LIN {X 0,Y 432.916,Z 623.479,A -85,B 0,C 180,E1 19556.175,E2 19556.175} C_VEL
LIN {X 0,Y 430.996,Z 639.731,A -85,B 0,C 180,E1 19554.827,E2 19554.827} C_VEL
LIN {X 0,Y 428.968,Z 654.603,A -85,B 0,C 180,E1 19553.313,E2 19553.313} C_VEL
LIN {X 0,Y 426.86,Z 668.614,A -85,B 0,C 180,E1 19551.576,E2 19551.576} C_VEL
LIN {X 0,Y 424.795,Z 681.338,A -85,B 0,C 180,E1 19549.668,E2 19549.668} C_VEL
LIN {X 0,Y 422.892,Z 692.644,A -85,B 0,C 180,E1 19547.615,E2 19547.615} C_VEL
LIN {X 0,Y 421.141,Z 703.114,A -85,B 0,C 180,E1 19545.279,E2 19545.279} C_VEL
LIN {X 0,Y 419.749,Z 711.572,A -85,B 0,C 180,E1 19542.939,E2 19542.939} C_VEL
LIN {X 0,Y 418.624,Z 718.946,A -85,B 0,C 180,E1 19540.319,E2 19540.319} C_VEL
LIN {X 0,Y 417.88,Z 724.436,A -85,B 0,C 180,E1 19537.7,E2 19537.7} C_VEL
LIN {X 0,Y 417.414,Z 728.221,A -85,B 0,C 180,E1 19535.085,E2 19535.085} C_VEL
LIN {X 0,Y 417.168,Z 730.486,A -85,B 0,C 180,E1 19532.335,E2 19532.335} C_VEL
LIN {X 0,Y 417.109,Z 731.085,A -85,B 0,C 180,E1 19529.588,E2 19529.588} C_VEL
LIN {X 0,Y 417.21,Z 730.043,A -85,B 0,C 180,E1 19526.84,E2 19526.84} C_VEL
LIN {X 0,Y 417.516,Z 727.312,A -85,B 0,C 180,E1 19524.09,E2 19524.09} C_VEL
LIN {X 0,Y 418.1,Z 722.784,A -85,B 0,C 180,E1 19521.335,E2 19521.335} C_VEL
LIN {X 0,Y 418.949,Z 716.685,A -85,B 0,C 180,E1 19518.715,E2 19518.715} C_VEL
LIN {X 0,Y 420.139,Z 709.085,A -85,B 0,C 180,E1 19516.233,E2 19516.233} C_VEL
LIN {X 0,Y 421.646,Z 700.029,A -85,B 0,C 180,E1 19513.893,E2 19513.893} C_VEL
LIN {X 0,Y 423.426,Z 689.42,A -85,B 0,C 180,E1 19511.672,E2 19511.672} C_VEL
LIN {X 0,Y 425.411,Z 677.603,A -85,B 0,C 180,E1 19509.645,E2 19509.645} C_VEL
LIN {X 0,Y 427.552,Z 664.114,A -85,B 0,C 180,E1 19507.738,E2 19507.738} C_VEL
LIN {X 0,Y 429.701,Z 649.518,A -85,B 0,C 180,E1 19506.045,E2 19506.045} C_VEL
LIN {X 0,Y 431.738,Z 633.856,A -85,B 0,C 180,E1 19504.559,E2 19504.559} C_VEL
LIN {X 0,Y 433.596,Z 617.11,A -85,B 0,C 180,E1 19503.279,E2 19503.279} C_VEL
LIN {X 0,Y 435.079,Z 600.265,A -85,B 0,C 180,E1 19502.26,E2 19502.26} C_VEL
LIN {X 0,Y 436.268,Z 581.748,A -85,B 0,C 180,E1 19501.409,E2 19501.409} C_VEL
LIN {X 0,Y 436.995,Z 563.024,A -85,B 0,C 180,E1 19500.806,E2 19500.806} C_VEL
LIN {X 0,Y 437.369,Z 538.708,A -85,B 0,C 180,E1 19500.338,E2 19500.338} C_VEL
LIN {X 0,Y 440.401,Z 366.683,A -85,B 0,C 180,E1 19497.558,E2 19497.558} C_VEL
LIN {X 0,Y 438.664,Z 359.169,A -85,B 0,C 180,E1 19497.254,E2 19497.254} C_VEL
LIN {X 0,Y 429.753,Z 342.969,A -85,B 0,C 180,E1 19496.041,E2 19496.041} C_VEL
LIN {X 0,Y 423.803,Z 326.84,A -85,B 0,C 180,E1 19493.336,E2 19493.336} C_VEL
LIN {X 0,Y 418.468,Z 313.652,A -85,B 0,C 180,E1 19490.893,E2 19490.893} C_VEL
LIN {X 0,Y 417.399,Z 310.595,A -85,B 0,C 180,E1 19490.241,E2 19490.241} C_VEL
LIN {X 0,Y 417.367,Z 310.446,A -85,B 0,C 180,E1 19486.343,E2 19486.343} C_VEL
LIN {X 0,Y 417.361,Z 310.494,A -85,B 0,C 180,E1 19482.452,E2 19482.452} C_VEL
LIN {X 0,Y 417.347,Z 310.491,A -85,B 0,C 180,E1 19478.649,E2 19478.649} C_VEL
LIN {X 0,Y 417.341,Z 310.491,A -85,B 0,C 180,E1 19474.764,E2 19474.764} C_VEL
LIN {X 0,Y 417.335,Z 310.495,A -85,B 0,C 180,E1 19470.845,E2 19470.845} C_VEL
LIN {X 0,Y 417.335,Z 310.499,A -85,B 0,C 180,E1 19466.924,E2 19466.924} C_VEL
LIN {X 0,Y 417.336,Z 310.498,A -85,B 0,C 180,E1 19463.079,E2 19463.079} C_VEL
LIN {X 0,Y 417.355,Z 310.477,A -85,B 0,C 180,E1 19459.451,E2 19459.451} C_VEL
LIN {X 0,Y 417.368,Z 310.483,A -85,B 0,C 180,E1 19455.564,E2 19455.564} C_VEL
LIN {X 0,Y 417.358,Z 310.496,A -85,B 0,C 180,E1 19451.75,E2 19451.75} C_VEL
LIN {X 0,Y 417.343,Z 310.478,A -85,B 0,C 180,E1 19447.849,E2 19447.849} C_VEL
LIN {X 0,Y 417.317,Z 310.49,A -85,B 0,C 180,E1 19444.122,E2 19444.122} C_VEL
LIN {X 0,Y 417.302,Z 310.501,A -85,B 0,C 180,E1 19440.412,E2 19440.412} C_VEL
LIN {X 0,Y 417.303,Z 310.484,A -85,B 0,C 180,E1 19436.566,E2 19436.566} C_VEL
LIN {X 0,Y 417.318,Z 310.487,A -85,B 0,C 180,E1 19432.843,E2 19432.843} C_VEL
LIN {X 0,Y 417.345,Z 310.499,A -85,B 0,C 180,E1 19429.09,E2 19429.09} C_VEL
LIN {X 0,Y 417.373,Z 310.483,A -85,B 0,C 180,E1 19425.29,E2 19425.29} C_VEL
LIN {X 0,Y 417.364,Z 310.479,A -85,B 0,C 180,E1 19421.421,E2 19421.421} C_VEL
LIN {X 0,Y 417.353,Z 310.485,A -85,B 0,C 180,E1 19417.61,E2 19417.61} C_VEL
LIN {X 0,Y 417.34,Z 310.493,A -85,B 0,C 180,E1 19413.844,E2 19413.844} C_VEL
LIN {X 0,Y 417.334,Z 310.497,A -85,B 0,C 180,E1 19410.111,E2 19410.111} C_VEL
LIN {X 0,Y 417.337,Z 310.486,A -85,B 0,C 180,E1 19406.233,E2 19406.233} C_VEL
LIN {X 0,Y 417.341,Z 310.465,A -85,B 0,C 180,E1 19402.344,E2 19402.344} C_VEL
LIN {X 0,Y 417.358,Z 310.451,A -85,B 0,C 180,E1 19398.608,E2 19398.608} C_VEL
LIN {X 0,Y 417.389,Z 310.785,A -85,B 0,C 180,E1 19398.001,E2 19398.001} C_VEL
LIN {X 0,Y 418.612,Z 313.856,A -85,B 0,C 180,E1 19397.472,E2 19397.472} C_VEL
LIN {X 0,Y 425.196,Z 327.627,A -85,B 0,C 180,E1 19395.324,E2 19395.324} C_VEL
LIN {X 0,Y 433.412,Z 346.345,A -85,B 0,C 180,E1 19392.705,E2 19392.705} C_VEL
LIN {X 0,Y 439.742,Z 362.777,A -85,B 0,C 180,E1 19390.648,E2 19390.648} C_VEL
LIN {X 0,Y 437.871,Z 383.994,A -85,B 0,C 180,E1 19389.058,E2 19389.058} C_VEL
LIN {X 0,Y 441.536,Z 419.357,A -85,B 0,C 180,E1 19387.995,E2 19387.995} C_VEL
LIN {X 0,Y 435.739,Z 636.384,A -85,B 0,C 180,E1 19384.015,E2 19384.015} C_VEL
LIN {X 0,Y 434.519,Z 657.893,A -85,B 0,C 180,E1 19383.442,E2 19383.442} C_VEL
LIN {X 0,Y 432.751,Z 679.3,A -85,B 0,C 180,E1 19382.622,E2 19382.622} C_VEL
LIN {X 0,Y 430.784,Z 699.969,A -85,B 0,C 180,E1 19381.559,E2 19381.559} C_VEL
LIN {X 0,Y 428.751,Z 719.018,A -85,B 0,C 180,E1 19380.323,E2 19380.323} C_VEL
LIN {X 0,Y 426.668,Z 737.44,A -85,B 0,C 180,E1 19378.864,E2 19378.864} C_VEL
LIN {X 0,Y 424.603,Z 755.114,A -85,B 0,C 180,E1 19377.182,E2 19377.182} C_VEL
LIN {X 0,Y 422.491,Z 773.079,A -85,B 0,C 180,E1 19375.137,E2 19375.137} C_VEL
LIN {X 0,Y 420.637,Z 789.749,A -85,B 0,C 180,E1 19372.869,E2 19372.869} C_VEL
LIN {X 0,Y 419.154,Z 804.214,A -85,B 0,C 180,E1 19370.527,E2 19370.527} C_VEL
LIN {X 0,Y 418.029,Z 816.771,A -85,B 0,C 180,E1 19368.115,E2 19368.115} C_VEL
LIN {X 0,Y 417.232,Z 827.882,A -85,B 0,C 180,E1 19365.568,E2 19365.568} C_VEL
LIN {X 0,Y 416.703,Z 837.456,A -85,B 0,C 180,E1 19362.894,E2 19362.894} C_VEL
LIN {X 0,Y 416.453,Z 845.052,A -85,B 0,C 180,E1 19360.234,E2 19360.234} C_VEL
LIN {X 0,Y 416.366,Z 850.572,A -85,B 0,C 180,E1 19357.728,E2 19357.728} C_VEL
LIN {X 0,Y 416.386,Z 854.593,A -85,B 0,C 180,E1 19355.097,E2 19355.097} C_VEL
LIN {X 0,Y 416.426,Z 856.966,A -85,B 0,C 180,E1 19352.477,E2 19352.477} C_VEL
LIN {X 0,Y 416.447,Z 857.743,A -85,B 0,C 180,E1 19349.862,E2 19349.862} C_VEL
LIN {X 0,Y 416.427,Z 856.813,A -85,B 0,C 180,E1 19347.248,E2 19347.248} C_VEL
LIN {X 0,Y 416.387,Z 854.237,A -85,B 0,C 180,E1 19344.627,E2 19344.627} C_VEL
LIN {X 0,Y 416.374,Z 850.01,A -85,B 0,C 180,E1 19341.994,E2 19341.994} C_VEL
LIN {X 0,Y 416.483,Z 844.036,A -85,B 0,C 180,E1 19339.348,E2 19339.348} C_VEL
LIN {X 0,Y 416.764,Z 836.113,A -85,B 0,C 180,E1 19336.685,E2 19336.685} C_VEL
LIN {X 0,Y 417.308,Z 826.752,A -85,B 0,C 180,E1 19334.149,E2 19334.149} C_VEL
LIN {X 0,Y 418.148,Z 815.386,A -85,B 0,C 180,E1 19331.602,E2 19331.602} C_VEL
LIN {X 0,Y 419.315,Z 802.509,A -85,B 0,C 180,E1 19329.183,E2 19329.183} C_VEL
LIN {X 0,Y 420.797,Z 788.255,A -85,B 0,C 180,E1 19326.918,E2 19326.918} C_VEL
LIN {X 0,Y 422.553,Z 772.476,A -85,B 0,C 180,E1 19324.792,E2 19324.792} C_VEL
LIN {X 0,Y 424.601,Z 755.097,A -85,B 0,C 180,E1 19322.818,E2 19322.818} C_VEL
LIN {X 0,Y 426.762,Z 736.64,A -85,B 0,C 180,E1 19321.067,E2 19321.067} C_VEL
LIN {X 0,Y 428.972,Z 717.108,A -85,B 0,C 180,E1 19319.54,E2 19319.54} C_VEL
LIN {X 0,Y 431.019,Z 697.589,A -85,B 0,C 180,E1 19318.304,E2 19318.304} C_VEL
LIN {X 0,Y 432.834,Z 678.286,A -85,B 0,C 180,E1 19317.335,E2 19317.335} C_VEL
LIN {X 0,Y 434.552,Z 657.279,A -85,B 0,C 180,E1 19316.541,E2 19316.541} C_VEL
LIN {X 0,Y 435.772,Z 635.074,A -85,B 0,C 180,E1 19315.961,E2 19315.961} C_VEL
LIN {X 0,Y 441.555,Z 417.909,A -85,B 0,C 180,E1 19311.983,E2 19311.983} C_VEL
LIN {X 0,Y 437.832,Z 382.808,A -85,B 0,C 180,E1 19310.888,E2 19310.888} C_VEL
LIN {X 0,Y 439.679,Z 362.43,A -85,B 0,C 180,E1 19309.323,E2 19309.323} C_VEL
LIN {X 0,Y 431.887,Z 342.744,A -85,B 0,C 180,E1 19306.824,E2 19306.824} C_VEL
LIN {X 0,Y 423.924,Z 324.867,A -85,B 0,C 180,E1 19304.278,E2 19304.278} C_VEL
LIN {X 0,Y 419.049,Z 314.463,A -85,B 0,C 180,E1 19302.658,E2 19302.658} C_VEL
LIN {X 0,Y 417.415,Z 310.928,A -85,B 0,C 180,E1 19302.052,E2 19302.052} C_VEL
LIN {X 0,Y 417.349,Z 310.452,A -85,B 0,C 180,E1 19301.576,E2 19301.576} C_VEL
LIN {X 0,Y 417.34,Z 310.47,A -85,B 0,C 180,E1 19297.83,E2 19297.83} C_VEL
LIN {X 0,Y 417.339,Z 310.481,A -85,B 0,C 180,E1 19293.932,E2 19293.932} C_VEL
LIN {X 0,Y 417.341,Z 310.495,A -85,B 0,C 180,E1 19290.047,E2 19290.047} C_VEL
LIN {X 0,Y 417.351,Z 310.49,A -85,B 0,C 180,E1 19286.309,E2 19286.309} C_VEL
LIN {X 0,Y 417.369,Z 310.482,A -85,B 0,C 180,E1 19282.538,E2 19282.538} C_VEL
LIN {X 0,Y 417.371,Z 310.479,A -85,B 0,C 180,E1 19278.724,E2 19278.724} C_VEL
LIN {X 0,Y 417.36,Z 310.488,A -85,B 0,C 180,E1 19274.853,E2 19274.853} C_VEL
LIN {X 0,Y 417.336,Z 310.499,A -85,B 0,C 180,E1 19271.05,E2 19271.05} C_VEL
LIN {X 0,Y 417.316,Z 310.489,A -85,B 0,C 180,E1 19267.295,E2 19267.295} C_VEL
LIN {X 0,Y 417.307,Z 310.487,A -85,B 0,C 180,E1 19263.571,E2 19263.571} C_VEL
LIN {X 0,Y 417.308,Z 310.502,A -85,B 0,C 180,E1 19259.725,E2 19259.725} C_VEL
LIN {X 0,Y 417.322,Z 310.486,A -85,B 0,C 180,E1 19256.016,E2 19256.016} C_VEL
LIN {X 0,Y 417.355,Z 310.478,A -85,B 0,C 180,E1 19252.29,E2 19252.29} C_VEL
LIN {X 0,Y 417.357,Z 310.5,A -85,B 0,C 180,E1 19248.39,E2 19248.39} C_VEL
LIN {X 0,Y 417.349,Z 310.483,A -85,B 0,C 180,E1 19244.578,E2 19244.578} C_VEL
LIN {X 0,Y 417.33,Z 310.482,A -85,B 0,C 180,E1 19240.838,E2 19240.838} C_VEL
LIN {X 0,Y 417.324,Z 310.5,A -85,B 0,C 180,E1 19237.161,E2 19237.161} C_VEL
LIN {X 0,Y 417.328,Z 310.499,A -85,B 0,C 180,E1 19233.229,E2 19233.229} C_VEL
LIN {X 0,Y 417.333,Z 310.494,A -85,B 0,C 180,E1 19229.325,E2 19229.325} C_VEL
LIN {X 0,Y 417.344,Z 310.488,A -85,B 0,C 180,E1 19225.499,E2 19225.499} C_VEL
LIN {X 0,Y 417.37,Z 310.484,A -85,B 0,C 180,E1 19221.789,E2 19221.789} C_VEL
LIN {X 0,Y 417.382,Z 310.485,A -85,B 0,C 180,E1 19217.953,E2 19217.953} C_VEL
LIN {X 0,Y 417.375,Z 310.446,A -85,B 0,C 180,E1 19214.054,E2 19214.054} C_VEL
LIN {X 0,Y 417.381,Z 310.473,A -85,B 0,C 180,E1 19210.12,E2 19210.12} C_VEL
LIN {X 0,Y 417.423,Z 310.821,A -85,B 0,C 180,E1 19209.56,E2 19209.56} C_VEL
LIN {X 0,Y 423.284,Z 325.515,A -85,B 0,C 180,E1 19206.796,E2 19206.796} C_VEL
LIN {X 0,Y 429.434,Z 342.168,A -85,B 0,C 180,E1 19203.971,E2 19203.971} C_VEL
LIN {X 0,Y 430.778,Z 344.992,A -85,B 0,C 180,E1 19203.685,E2 19203.685} C_VEL
LIN {X 0,Y 439.064,Z 360.282,A -85,B 0,C 180,E1 19202.586,E2 19202.586} C_VEL
LIN {X 0,Y 440.446,Z 368.261,A -85,B 0,C 180,E1 19202.307,E2 19202.307} C_VEL
LIN {X 0,Y 437.093,Z 558.617,A -85,B 0,C 180,E1 19199.21,E2 19199.21} C_VEL
LIN {X 0,Y 436.455,Z 577.921,A -85,B 0,C 180,E1 19198.644,E2 19198.644} C_VEL
LIN {X 0,Y 435.833,Z 589.062,A -85,B 0,C 180,E1 19198.193,E2 19198.193} C_VEL
LIN {X 0,Y 434.477,Z 596.631,A -85,B 0,C 180,E1 19197.912,E2 19197.912} C_VEL
LIN {X 0,Y 428.112,Z 614.037,A -85,B 0,C 180,E1 19197.327,E2 19197.327} C_VEL
LIN {X 0,Y 426.369,Z 620.792,A -85,B 0,C 180,E1 19196.95,E2 19196.95} C_VEL
LIN {X 0,Y 426.252,Z 621.745,A -85,B 0,C 180,E1 19196.885,E2 19196.885} C_VEL
LIN {X 0,Y 424.256,Z 638.214,A -85,B 0,C 180,E1 19195.548,E2 19195.548} C_VEL
LIN {X 0,Y 422.152,Z 653.265,A -85,B 0,C 180,E1 19194.04,E2 19194.04} C_VEL
LIN {X 0,Y 420.017,Z 666.865,A -85,B 0,C 180,E1 19192.388,E2 19192.388} C_VEL
LIN {X 0,Y 417.793,Z 680.072,A -85,B 0,C 180,E1 19190.45,E2 19190.45} C_VEL
LIN {X 0,Y 415.714,Z 691.783,A -85,B 0,C 180,E1 19188.365,E2 19188.365} C_VEL
LIN {X 0,Y 413.892,Z 702.067,A -85,B 0,C 180,E1 19186.129,E2 19186.129} C_VEL
LIN {X 0,Y 412.327,Z 710.951,A -85,B 0,C 180,E1 19183.747,E2 19183.747} C_VEL
LIN {X 0,Y 411.096,Z 718.401,A -85,B 0,C 180,E1 19181.22,E2 19181.22} C_VEL
LIN {X 0,Y 410.21,Z 724.366,A -85,B 0,C 180,E1 19178.55,E2 19178.55} C_VEL
LIN {X 0,Y 409.629,Z 728.578,A -85,B 0,C 180,E1 19175.884,E2 19175.884} C_VEL
LIN {X 0,Y 409.305,Z 731.277,A -85,B 0,C 180,E1 19173.081,E2 19173.081} C_VEL
LIN {X 0,Y 409.2,Z 732.293,A -85,B 0,C 180,E1 19170.28,E2 19170.28} C_VEL
LIN {X 0,Y 409.271,Z 731.67,A -85,B 0,C 180,E1 19167.48,E2 19167.48} C_VEL
LIN {X 0,Y 409.538,Z 729.386,A -85,B 0,C 180,E1 19164.677,E2 19164.677} C_VEL
LIN {X 0,Y 410.084,Z 725.347,A -85,B 0,C 180,E1 19161.871,E2 19161.871} C_VEL
LIN {X 0,Y 410.908,Z 719.743,A -85,B 0,C 180,E1 19159.201,E2 19159.201} C_VEL
LIN {X 0,Y 412.133,Z 712.22,A -85,B 0,C 180,E1 19156.532,E2 19156.532} C_VEL
LIN {X 0,Y 413.645,Z 703.643,A -85,B 0,C 180,E1 19154.149,E2 19154.149} C_VEL
LIN {X 0,Y 415.525,Z 692.986,A -85,B 0,C 180,E1 19151.772,E2 19151.772} C_VEL
LIN {X 0,Y 417.57,Z 681.528,A -85,B 0,C 180,E1 19149.685,E2 19149.685} C_VEL
LIN {X 0,Y 419.849,Z 668.093,A -85,B 0,C 180,E1 19147.677,E2 19147.677} C_VEL
LIN {X 0,Y 422.052,Z 654.11,A -85,B 0,C 180,E1 19145.954,E2 19145.954} C_VEL
LIN {X 0,Y 424.252,Z 638.461,A -85,B 0,C 180,E1 19144.377,E2 19144.377} C_VEL
LIN {X 0,Y 426.243,Z 622.169,A -85,B 0,C 180,E1 19143.049,E2 19143.049} C_VEL
LIN {X 0,Y 427.946,Z 604.675,A -85,B 0,C 180,E1 19141.916,E2 19141.916} C_VEL
LIN {X 0,Y 429.264,Z 586.618,A -85,B 0,C 180,E1 19141.022,E2 19141.022} C_VEL
LIN {X 0,Y 430.126,Z 567.98,A -85,B 0,C 180,E1 19140.359,E2 19140.359} C_VEL
LIN {X 0,Y 430.528,Z 548.32,A -85,B 0,C 180,E1 19139.919,E2 19139.919} C_VEL
LIN {X 0,Y 433.863,Z 368.04,A -85,B 0,C 180,E1 19136.96,E2 19136.96} C_VEL
LIN {X 0,Y 432.581,Z 362.846,A -85,B 0,C 180,E1 19136.736,E2 19136.736} C_VEL
LIN {X 0,Y 421.819,Z 343.427,A -85,B 0,C 180,E1 19135.218,E2 19135.218} C_VEL
LIN {X 0,Y 415.921,Z 327.808,A -85,B 0,C 180,E1 19132.496,E2 19132.496} C_VEL
LIN {X 0,Y 410.61,Z 314.728,A -85,B 0,C 180,E1 19129.996,E2 19129.996} C_VEL
LIN {X 0,Y 409.438,Z 311.625,A -85,B 0,C 180,E1 19129.307,E2 19129.307} C_VEL
LIN {X 0,Y 409.42,Z 311.437,A -85,B 0,C 180,E1 19125.488,E2 19125.488} C_VEL
LIN {X 0,Y 409.436,Z 311.472,A -85,B 0,C 180,E1 19121.624,E2 19121.624} C_VEL
LIN {X 0,Y 409.442,Z 311.47,A -85,B 0,C 180,E1 19117.803,E2 19117.803} C_VEL
LIN {X 0,Y 409.438,Z 311.468,A -85,B 0,C 180,E1 19113.834,E2 19113.834} C_VEL
LIN {X 0,Y 409.449,Z 311.466,A -85,B 0,C 180,E1 19109.879,E2 19109.879} C_VEL
LIN {X 0,Y 409.43,Z 311.474,A -85,B 0,C 180,E1 19105.921,E2 19105.921} C_VEL
LIN {X 0,Y 409.415,Z 311.487,A -85,B 0,C 180,E1 19102.092,E2 19102.092} C_VEL
LIN {X 0,Y 409.398,Z 311.479,A -85,B 0,C 180,E1 19098.217,E2 19098.217} C_VEL
LIN {X 0,Y 409.381,Z 311.466,A -85,B 0,C 180,E1 19094.426,E2 19094.426} C_VEL
LIN {X 0,Y 409.377,Z 311.487,A -85,B 0,C 180,E1 19090.555,E2 19090.555} C_VEL
LIN {X 0,Y 409.37,Z 311.489,A -85,B 0,C 180,E1 19086.592,E2 19086.592} C_VEL
LIN {X 0,Y 409.364,Z 311.468,A -85,B 0,C 180,E1 19082.64,E2 19082.64} C_VEL
LIN {X 0,Y 409.372,Z 311.482,A -85,B 0,C 180,E1 19078.881,E2 19078.881} C_VEL
LIN {X 0,Y 409.394,Z 311.487,A -85,B 0,C 180,E1 19075.097,E2 19075.097} C_VEL
LIN {X 0,Y 409.416,Z 311.465,A -85,B 0,C 180,E1 19071.291,E2 19071.291} C_VEL
LIN {X 0,Y 409.422,Z 311.467,A -85,B 0,C 180,E1 19067.304,E2 19067.304} C_VEL
LIN {X 0,Y 409.429,Z 311.483,A -85,B 0,C 180,E1 19063.398,E2 19063.398} C_VEL
LIN {X 0,Y 409.429,Z 311.486,A -85,B 0,C 180,E1 19059.411,E2 19059.411} C_VEL
LIN {X 0,Y 409.413,Z 311.481,A -85,B 0,C 180,E1 19055.624,E2 19055.624} C_VEL
LIN {X 0,Y 409.404,Z 311.479,A -85,B 0,C 180,E1 19051.838,E2 19051.838} C_VEL
LIN {X 0,Y 409.4,Z 311.482,A -85,B 0,C 180,E1 19047.997,E2 19047.997} C_VEL
LIN {X 0,Y 409.395,Z 311.433,A -85,B 0,C 180,E1 19044.116,E2 19044.116} C_VEL
LIN {X 0,Y 409.404,Z 311.469,A -85,B 0,C 180,E1 19040.219,E2 19040.219} C_VEL
LIN {X 0,Y 409.488,Z 311.753,A -85,B 0,C 180,E1 19038.979,E2 19038.979} C_VEL
LIN {X 0,Y 410.878,Z 315.161,A -85,B 0,C 180,E1 19038.369,E2 19038.369} C_VEL
LIN {X 0,Y 417.354,Z 328.537,A -85,B 0,C 180,E1 19036.183,E2 19036.183} C_VEL
LIN {X 0,Y 425.615,Z 347.272,A -85,B 0,C 180,E1 19033.456,E2 19033.456} C_VEL
LIN {X 0,Y 432.84,Z 365.718,A -85,B 0,C 180,E1 19031.063,E2 19031.063} C_VEL
LIN {X 0,Y 431.181,Z 383.563,A -85,B 0,C 180,E1 19029.707,E2 19029.707} C_VEL
LIN {X 0,Y 434.934,Z 420.487,A -85,B 0,C 180,E1 19028.574,E2 19028.574} C_VEL
LIN {X 0,Y 428.868,Z 635.975,A -85,B 0,C 180,E1 19024.566,E2 19024.566} C_VEL
LIN {X 0,Y 427.59,Z 657.284,A -85,B 0,C 180,E1 19023.986,E2 19023.986} C_VEL
LIN {X 0,Y 425.77,Z 678.267,A -85,B 0,C 180,E1 19023.172,E2 19023.172} C_VEL
LIN {X 0,Y 423.67,Z 699.069,A -85,B 0,C 180,E1 19022.088,E2 19022.088} C_VEL
LIN {X 0,Y 421.507,Z 718.264,A -85,B 0,C 180,E1 19020.821,E2 19020.821} C_VEL
LIN {X 0,Y 419.298,Z 736.613,A -85,B 0,C 180,E1 19019.342,E2 19019.342} C_VEL
LIN {X 0,Y 417.021,Z 754.9,A -85,B 0,C 180,E1 19017.563,E2 19017.563} C_VEL
LIN {X 0,Y 414.87,Z 772.149,A -85,B 0,C 180,E1 19015.556,E2 19015.556} C_VEL
LIN {X 0,Y 412.957,Z 788.311,A -85,B 0,C 180,E1 19013.315,E2 19013.315} C_VEL
LIN {X 0,Y 411.362,Z 802.783,A -85,B 0,C 180,E1 19010.934,E2 19010.934} C_VEL
LIN {X 0,Y 410.167,Z 815.378,A -85,B 0,C 180,E1 19008.475,E2 19008.475} C_VEL
LIN {X 0,Y 409.313,Z 826.523,A -85,B 0,C 180,E1 19005.878,E2 19005.878} C_VEL
LIN {X 0,Y 408.754,Z 836.131,A -85,B 0,C 180,E1 19003.149,E2 19003.149} C_VEL
LIN {X 0,Y 408.506,Z 843.761,A -85,B 0,C 180,E1 19000.435,E2 19000.435} C_VEL
LIN {X 0,Y 408.424,Z 849.304,A -85,B 0,C 180,E1 18997.879,E2 18997.879} C_VEL
LIN {X 0,Y 408.46,Z 853.36,A -85,B 0,C 180,E1 18995.196,E2 18995.196} C_VEL
LIN {X 0,Y 408.514,Z 855.759,A -85,B 0,C 180,E1 18992.525,E2 18992.525} C_VEL
LIN {X 0,Y 408.54,Z 856.558,A -85,B 0,C 180,E1 18990,E2 18990} C_VEL
LIN {X 0,Y 408.515,Z 855.681,A -85,B 0,C 180,E1 18987.335,E2 18987.335} C_VEL
LIN {X 0,Y 408.462,Z 853.181,A -85,B 0,C 180,E1 18984.663,E2 18984.663} C_VEL
LIN {X 0,Y 408.429,Z 849.023,A -85,B 0,C 180,E1 18981.979,E2 18981.979} C_VEL
LIN {X 0,Y 408.516,Z 843.427,A -85,B 0,C 180,E1 18979.423,E2 18979.423} C_VEL
LIN {X 0,Y 408.765,Z 835.93,A -85,B 0,C 180,E1 18976.786,E2 18976.786} C_VEL
LIN {X 0,Y 409.313,Z 826.523,A -85,B 0,C 180,E1 18974.122,E2 18974.122} C_VEL
LIN {X 0,Y 410.167,Z 815.376,A -85,B 0,C 180,E1 18971.525,E2 18971.525} C_VEL
LIN {X 0,Y 411.364,Z 802.779,A -85,B 0,C 180,E1 18969.066,E2 18969.066} C_VEL
LIN {X 0,Y 412.956,Z 788.304,A -85,B 0,C 180,E1 18966.685,E2 18966.685} C_VEL
LIN {X 0,Y 414.868,Z 772.131,A -85,B 0,C 180,E1 18964.444,E2 18964.444} C_VEL
LIN {X 0,Y 417.103,Z 754.217,A -85,B 0,C 180,E1 18962.365,E2 18962.365} C_VEL
LIN {X 0,Y 419.395,Z 735.81,A -85,B 0,C 180,E1 18960.587,E2 18960.587} C_VEL
LIN {X 0,Y 421.736,Z 716.344,A -85,B 0,C 180,E1 18959.039,E2 18959.039} C_VEL
LIN {X 0,Y 423.888,Z 696.913,A -85,B 0,C 180,E1 18957.787,E2 18957.787} C_VEL
LIN {X 0,Y 425.839,Z 677.437,A -85,B 0,C 180,E1 18956.794,E2 18956.794} C_VEL
LIN {X 0,Y 427.644,Z 656.33,A -85,B 0,C 180,E1 18955.986,E2 18955.986} C_VEL
LIN {X 0,Y 428.917,Z 634.217,A -85,B 0,C 180,E1 18955.401,E2 18955.401} C_VEL
LIN {X 0,Y 434.949,Z 419.079,A -85,B 0,C 180,E1 18951.405,E2 18951.405} C_VEL
LIN {X 0,Y 431.128,Z 382.442,A -85,B 0,C 180,E1 18950.245,E2 18950.245} C_VEL
LIN {X 0,Y 432.662,Z 365.234,A -85,B 0,C 180,E1 18948.883,E2 18948.883} C_VEL
LIN {X 0,Y 424.953,Z 345.751,A -85,B 0,C 180,E1 18946.344,E2 18946.344} C_VEL
LIN {X 0,Y 416.913,Z 327.6,A -85,B 0,C 180,E1 18943.685,E2 18943.685} C_VEL
LIN {X 0,Y 410.84,Z 315.109,A -85,B 0,C 180,E1 18941.636,E2 18941.636} C_VEL
LIN {X 0,Y 409.479,Z 311.692,A -85,B 0,C 180,E1 18941.019,E2 18941.019} C_VEL
LIN {X 0,Y 409.431,Z 311.437,A -85,B 0,C 180,E1 18937.098,E2 18937.098} C_VEL
LIN {X 0,Y 409.427,Z 311.484,A -85,B 0,C 180,E1 18933.163,E2 18933.163} C_VEL
LIN {X 0,Y 409.412,Z 311.489,A -85,B 0,C 180,E1 18929.328,E2 18929.328} C_VEL
LIN {X 0,Y 409.395,Z 311.49,A -85,B 0,C 180,E1 18925.612,E2 18925.612} C_VEL
LIN {X 0,Y 409.389,Z 311.485,A -85,B 0,C 180,E1 18921.791,E2 18921.791} C_VEL
LIN {X 0,Y 409.389,Z 311.474,A -85,B 0,C 180,E1 18917.922,E2 18917.922} C_VEL
LIN {X 0,Y 409.395,Z 311.468,A -85,B 0,C 180,E1 18914.136,E2 18914.136} C_VEL
LIN {X 0,Y 409.405,Z 311.484,A -85,B 0,C 180,E1 18910.269,E2 18910.269} C_VEL
LIN {X 0,Y 409.423,Z 311.48,A -85,B 0,C 180,E1 18906.45,E2 18906.45} C_VEL
LIN {X 0,Y 409.413,Z 311.464,A -85,B 0,C 180,E1 18902.519,E2 18902.519} C_VEL
LIN {X 0,Y 409.397,Z 311.481,A -85,B 0,C 180,E1 18898.74,E2 18898.74} C_VEL
LIN {X 0,Y 409.389,Z 311.486,A -85,B 0,C 180,E1 18894.815,E2 18894.815} C_VEL
LIN {X 0,Y 409.37,Z 311.466,A -85,B 0,C 180,E1 18891.148,E2 18891.148} C_VEL
LIN {X 0,Y 409.372,Z 311.487,A -85,B 0,C 180,E1 18887.301,E2 18887.301} C_VEL
LIN {X 0,Y 409.38,Z 311.488,A -85,B 0,C 180,E1 18883.396,E2 18883.396} C_VEL
LIN {X 0,Y 409.386,Z 311.473,A -85,B 0,C 180,E1 18879.558,E2 18879.558} C_VEL
LIN {X 0,Y 409.415,Z 311.468,A -85,B 0,C 180,E1 18875.93,E2 18875.93} C_VEL
LIN {X 0,Y 409.434,Z 311.48,A -85,B 0,C 180,E1 18872.038,E2 18872.038} C_VEL
LIN {X 0,Y 409.442,Z 311.486,A -85,B 0,C 180,E1 18868.165,E2 18868.165} C_VEL
LIN {X 0,Y 409.438,Z 311.488,A -85,B 0,C 180,E1 18864.167,E2 18864.167} C_VEL
LIN {X 0,Y 409.441,Z 311.487,A -85,B 0,C 180,E1 18860.222,E2 18860.222} C_VEL
LIN {X 0,Y 409.432,Z 311.48,A -85,B 0,C 180,E1 18856.282,E2 18856.282} C_VEL
LIN {X 0,Y 409.423,Z 311.449,A -85,B 0,C 180,E1 18852.377,E2 18852.377} C_VEL
LIN {X 0,Y 409.445,Z 311.68,A -85,B 0,C 180,E1 18850.554,E2 18850.554} C_VEL
LIN {X 0,Y 414.039,Z 322.964,A -85,B 0,C 180,E1 18848.294,E2 18848.294} C_VEL
LIN {X 0,Y 420.183,Z 338.961,A -85,B 0,C 180,E1 18845.412,E2 18845.412} C_VEL
LIN {X 0,Y 422.114,Z 344.155,A -85,B 0,C 180,E1 18844.601,E2 18844.601} C_VEL
LIN {X 0,Y 432.944,Z 363.641,A -85,B 0,C 180,E1 18843.111,E2 18843.111} C_VEL
LIN {X 0,Y 433.926,Z 369.853,A -85,B 0,C 180,E1 18842.897,E2 18842.897} C_VEL
LIN {X 0,Y 430.344,Z 559.389,A -85,B 0,C 180,E1 18839.769,E2 18839.769} C_VEL
LIN {X 0,Y 429.672,Z 578.718,A -85,B 0,C 180,E1 18839.195,E2 18839.195} C_VEL
LIN {X 0,Y 428.534,Z 597.005,A -85,B 0,C 180,E1 18838.403,E2 18838.403} C_VEL
LIN {X 0,Y 427.032,Z 614.436,A -85,B 0,C 180,E1 18837.392,E2 18837.392} C_VEL
LIN {X 0,Y 426.252,Z 621.745,A -85,B 0,C 180,E1 18836.885,E2 18836.885} C_VEL
LIN {X 0,Y 424.656,Z 628.618,A -85,B 0,C 180,E1 18836.446,E2 18836.446} C_VEL
LIN {X 0,Y 417.575,Z 644.654,A -85,B 0,C 180,E1 18835.446,E2 18835.446} C_VEL
LIN {X 0,Y 415.555,Z 650.949,A -85,B 0,C 180,E1 18834.887,E2 18834.887} C_VEL
LIN {X 0,Y 415.401,Z 651.806,A -85,B 0,C 180,E1 18834.795,E2 18834.795} C_VEL
LIN {X 0,Y 412.991,Z 666.63,A -85,B 0,C 180,E1 18833.016,E2 18833.016} C_VEL
LIN {X 0,Y 410.554,Z 680.506,A -85,B 0,C 180,E1 18830.977,E2 18830.977} C_VEL
LIN {X 0,Y 408.344,Z 692.341,A -85,B 0,C 180,E1 18828.857,E2 18828.857} C_VEL
LIN {X 0,Y 406.394,Z 702.736,A -85,B 0,C 180,E1 18826.582,E2 18826.582} C_VEL
LIN {X 0,Y 404.717,Z 711.718,A -85,B 0,C 180,E1 18824.157,E2 18824.157} C_VEL
LIN {X 0,Y 403.38,Z 719.26,A -85,B 0,C 180,E1 18821.582,E2 18821.582} C_VEL
LIN {X 0,Y 402.414,Z 725.309,A -85,B 0,C 180,E1 18818.861,E2 18818.861} C_VEL
LIN {X 0,Y 401.778,Z 729.602,A -85,B 0,C 180,E1 18816.143,E2 18816.143} C_VEL
LIN {X 0,Y 401.414,Z 732.379,A -85,B 0,C 180,E1 18813.284,E2 18813.284} C_VEL
LIN {X 0,Y 401.291,Z 733.474,A -85,B 0,C 180,E1 18810.428,E2 18810.428} C_VEL
LIN {X 0,Y 401.356,Z 732.933,A -85,B 0,C 180,E1 18807.573,E2 18807.573} C_VEL
LIN {X 0,Y 401.632,Z 730.734,A -85,B 0,C 180,E1 18804.715,E2 18804.715} C_VEL
LIN {X 0,Y 402.161,Z 727.017,A -85,B 0,C 180,E1 18801.997,E2 18801.997} C_VEL
LIN {X 0,Y 403.008,Z 721.566,A -85,B 0,C 180,E1 18799.258,E2 18799.258} C_VEL
LIN {X 0,Y 404.18,Z 714.745,A -85,B 0,C 180,E1 18796.7,E2 18796.7} C_VEL
LIN {X 0,Y 405.709,Z 706.499,A -85,B 0,C 180,E1 18794.271,E2 18794.271} C_VEL
LIN {X 0,Y 407.496,Z 696.925,A -85,B 0,C 180,E1 18791.992,E2 18791.992} C_VEL
LIN {X 0,Y 409.545,Z 686.041,A -85,B 0,C 180,E1 18789.866,E2 18789.866} C_VEL
LIN {X 0,Y 411.773,Z 673.823,A -85,B 0,C 180,E1 18787.892,E2 18787.892} C_VEL
LIN {X 0,Y 414.185,Z 659.608,A -85,B 0,C 180,E1 18785.999,E2 18785.999} C_VEL
LIN {X 0,Y 416.559,Z 644.23,A -85,B 0,C 180,E1 18784.327,E2 18784.327} C_VEL
LIN {X 0,Y 418.648,Z 628.546,A -85,B 0,C 180,E1 18782.938,E2 18782.938} C_VEL
LIN {X 0,Y 420.602,Z 610.906,A -85,B 0,C 180,E1 18781.69,E2 18781.69} C_VEL
LIN {X 0,Y 422.101,Z 593.095,A -85,B 0,C 180,E1 18780.716,E2 18780.716} C_VEL
LIN {X 0,Y 423.186,Z 574.271,A -85,B 0,C 180,E1 18779.962,E2 18779.962} C_VEL
LIN {X 0,Y 423.733,Z 555.053,A -85,B 0,C 180,E1 18779.452,E2 18779.452} C_VEL
LIN {X 0,Y 427.381,Z 369.434,A -85,B 0,C 180,E1 18776.345,E2 18776.345} C_VEL
LIN {X 0,Y 426.448,Z 366.302,A -85,B 0,C 180,E1 18776.189,E2 18776.189} C_VEL
LIN {X 0,Y 414.197,Z 344.558,A -85,B 0,C 180,E1 18774.441,E2 18774.441} C_VEL
LIN {X 0,Y 408.67,Z 330.049,A -85,B 0,C 180,E1 18771.868,E2 18771.868} C_VEL
LIN {X 0,Y 402.76,Z 315.929,A -85,B 0,C 180,E1 18769.053,E2 18769.053} C_VEL
LIN {X 0,Y 401.525,Z 312.649,A -85,B 0,C 180,E1 18768.329,E2 18768.329} C_VEL
LIN {X 0,Y 401.478,Z 312.44,A -85,B 0,C 180,E1 18764.582,E2 18764.582} C_VEL
LIN {X 0,Y 401.468,Z 312.467,A -85,B 0,C 180,E1 18760.732,E2 18760.732} C_VEL
LIN {X 0,Y 401.464,Z 312.469,A -85,B 0,C 180,E1 18756.886,E2 18756.886} C_VEL
LIN {X 0,Y 401.46,Z 312.468,A -85,B 0,C 180,E1 18752.884,E2 18752.884} C_VEL
LIN {X 0,Y 401.461,Z 312.46,A -85,B 0,C 180,E1 18749.055,E2 18749.055} C_VEL
LIN {X 0,Y 401.464,Z 312.456,A -85,B 0,C 180,E1 18745.207,E2 18745.207} C_VEL
LIN {X 0,Y 401.472,Z 312.47,A -85,B 0,C 180,E1 18741.322,E2 18741.322} C_VEL
LIN {X 0,Y 401.475,Z 312.475,A -85,B 0,C 180,E1 18737.389,E2 18737.389} C_VEL
LIN {X 0,Y 401.485,Z 312.452,A -85,B 0,C 180,E1 18733.539,E2 18733.539} C_VEL
LIN {X 0,Y 401.478,Z 312.454,A -85,B 0,C 180,E1 18729.534,E2 18729.534} C_VEL
LIN {X 0,Y 401.473,Z 312.478,A -85,B 0,C 180,E1 18725.718,E2 18725.718} C_VEL
LIN {X 0,Y 401.463,Z 312.459,A -85,B 0,C 180,E1 18721.713,E2 18721.713} C_VEL
LIN {X 0,Y 401.446,Z 312.457,A -85,B 0,C 180,E1 18717.859,E2 18717.859} C_VEL
LIN {X 0,Y 401.445,Z 312.478,A -85,B 0,C 180,E1 18713.996,E2 18713.996} C_VEL
LIN {X 0,Y 401.44,Z 312.473,A -85,B 0,C 180,E1 18710.105,E2 18710.105} C_VEL
LIN {X 0,Y 401.439,Z 312.456,A -85,B 0,C 180,E1 18706.249,E2 18706.249} C_VEL
LIN {X 0,Y 401.443,Z 312.465,A -85,B 0,C 180,E1 18702.311,E2 18702.311} C_VEL
LIN {X 0,Y 401.45,Z 312.476,A -85,B 0,C 180,E1 18698.37,E2 18698.37} C_VEL
LIN {X 0,Y 401.457,Z 312.477,A -85,B 0,C 180,E1 18694.478,E2 18694.478} C_VEL
LIN {X 0,Y 401.472,Z 312.476,A -85,B 0,C 180,E1 18690.619,E2 18690.619} C_VEL
LIN {X 0,Y 401.482,Z 312.473,A -85,B 0,C 180,E1 18686.778,E2 18686.778} C_VEL
LIN {X 0,Y 401.487,Z 312.424,A -85,B 0,C 180,E1 18682.835,E2 18682.835} C_VEL
LIN {X 0,Y 401.483,Z 312.6,A -85,B 0,C 180,E1 18680.087,E2 18680.087} C_VEL
LIN {X 0,Y 401.977,Z 314.409,A -85,B 0,C 180,E1 18679.706,E2 18679.706} C_VEL
LIN {X 0,Y 403.647,Z 317.225,A -85,B 0,C 180,E1 18679.161,E2 18679.161} C_VEL
LIN {X 0,Y 411.959,Z 334.831,A -85,B 0,C 180,E1 18676.234,E2 18676.234} C_VEL
LIN {X 0,Y 419.94,Z 353.216,A -85,B 0,C 180,E1 18673.531,E2 18673.531} C_VEL
LIN {X 0,Y 425.942,Z 368.781,A -85,B 0,C 180,E1 18671.484,E2 18671.484} C_VEL
LIN {X 0,Y 424.548,Z 383.134,A -85,B 0,C 180,E1 18670.377,E2 18670.377} C_VEL
LIN {X 0,Y 428.38,Z 421.538,A -85,B 0,C 180,E1 18669.173,E2 18669.173} C_VEL
LIN {X 0,Y 422.048,Z 635.401,A -85,B 0,C 180,E1 18665.138,E2 18665.138} C_VEL
LIN {X 0,Y 420.712,Z 656.561,A -85,B 0,C 180,E1 18664.553,E2 18664.553} C_VEL
LIN {X 0,Y 418.852,Z 677.103,A -85,B 0,C 180,E1 18663.746,E2 18663.746} C_VEL
LIN {X 0,Y 416.672,Z 697.503,A -85,B 0,C 180,E1 18662.677,E2 18662.677} C_VEL
LIN {X 0,Y 414.42,Z 716.6,A -85,B 0,C 180,E1 18661.407,E2 18661.407} C_VEL
LIN {X 0,Y 412.063,Z 735.036,A -85,B 0,C 180,E1 18659.909,E2 18659.909} C_VEL
LIN {X 0,Y 409.64,Z 753.382,A -85,B 0,C 180,E1 18658.103,E2 18658.103} C_VEL
LIN {X 0,Y 407.343,Z 770.726,A -85,B 0,C 180,E1 18656.055,E2 18656.055} C_VEL
LIN {X 0,Y 405.274,Z 787.072,A -85,B 0,C 180,E1 18653.752,E2 18653.752} C_VEL
LIN {X 0,Y 403.568,Z 801.573,A -85,B 0,C 180,E1 18651.322,E2 18651.322} C_VEL
LIN {X 0,Y 402.31,Z 814.007,A -85,B 0,C 180,E1 18648.849,E2 18648.849} C_VEL
LIN {X 0,Y 401.391,Z 825.185,A -85,B 0,C 180,E1 18646.199,E2 18646.199} C_VEL
LIN {X 0,Y 400.807,Z 834.827,A -85,B 0,C 180,E1 18643.414,E2 18643.414} C_VEL
LIN {X 0,Y 400.554,Z 842.489,A -85,B 0,C 180,E1 18640.644,E2 18640.644} C_VEL
LIN {X 0,Y 400.48,Z 848.054,A -85,B 0,C 180,E1 18638.037,E2 18638.037} C_VEL
LIN {X 0,Y 400.534,Z 852.136,A -85,B 0,C 180,E1 18635.299,E2 18635.299} C_VEL
LIN {X 0,Y 400.6,Z 854.552,A -85,B 0,C 180,E1 18632.575,E2 18632.575} C_VEL
LIN {X 0,Y 400.631,Z 855.357,A -85,B 0,C 180,E1 18630,E2 18630} C_VEL
LIN {X 0,Y 400.601,Z 854.551,A -85,B 0,C 180,E1 18627.425,E2 18627.425} C_VEL
LIN {X 0,Y 400.534,Z 852.135,A -85,B 0,C 180,E1 18624.701,E2 18624.701} C_VEL
LIN {X 0,Y 400.481,Z 848.055,A -85,B 0,C 180,E1 18621.963,E2 18621.963} C_VEL
LIN {X 0,Y 400.554,Z 842.493,A -85,B 0,C 180,E1 18619.356,E2 18619.356} C_VEL
LIN {X 0,Y 400.808,Z 834.829,A -85,B 0,C 180,E1 18616.586,E2 18616.586} C_VEL
LIN {X 0,Y 401.392,Z 825.183,A -85,B 0,C 180,E1 18613.801,E2 18613.801} C_VEL
LIN {X 0,Y 402.31,Z 814.003,A -85,B 0,C 180,E1 18611.151,E2 18611.151} C_VEL
LIN {X 0,Y 403.587,Z 801.368,A -85,B 0,C 180,E1 18608.643,E2 18608.643} C_VEL
LIN {X 0,Y 405.27,Z 787.067,A -85,B 0,C 180,E1 18606.249,E2 18606.249} C_VEL
LIN {X 0,Y 407.34,Z 770.711,A -85,B 0,C 180,E1 18603.946,E2 18603.946} C_VEL
LIN {X 0,Y 409.638,Z 753.353,A -85,B 0,C 180,E1 18601.896,E2 18601.896} C_VEL
LIN {X 0,Y 412.059,Z 734.996,A -85,B 0,C 180,E1 18600.091,E2 18600.091} C_VEL
LIN {X 0,Y 414.537,Z 715.605,A -85,B 0,C 180,E1 18598.521,E2 18598.521} C_VEL
LIN {X 0,Y 416.797,Z 696.261,A -85,B 0,C 180,E1 18597.252,E2 18597.252} C_VEL
LIN {X 0,Y 418.842,Z 677.041,A -85,B 0,C 180,E1 18596.255,E2 18596.255} C_VEL
LIN {X 0,Y 420.754,Z 655.774,A -85,B 0,C 180,E1 18595.425,E2 18595.425} C_VEL
LIN {X 0,Y 422.094,Z 633.713,A -85,B 0,C 180,E1 18594.83,E2 18594.83} C_VEL
LIN {X 0,Y 428.393,Z 420.054,A -85,B 0,C 180,E1 18590.805,E2 18590.805} C_VEL
LIN {X 0,Y 424.501,Z 381.848,A -85,B 0,C 180,E1 18589.564,E2 18589.564} C_VEL
LIN {X 0,Y 425.87,Z 368.617,A -85,B 0,C 180,E1 18588.499,E2 18588.499} C_VEL
LIN {X 0,Y 418.455,Z 349.723,A -85,B 0,C 180,E1 18585.989,E2 18585.989} C_VEL
LIN {X 0,Y 410.699,Z 332.17,A -85,B 0,C 180,E1 18583.356,E2 18583.356} C_VEL
LIN {X 0,Y 404.68,Z 319.763,A -85,B 0,C 180,E1 18581.276,E2 18581.276} C_VEL
LIN {X 0,Y 403.187,Z 316.439,A -85,B 0,C 180,E1 18580.708,E2 18580.708} C_VEL
LIN {X 0,Y 401.523,Z 312.834,A -85,B 0,C 180,E1 18580.034,E2 18580.034} C_VEL
LIN {X 0,Y 401.471,Z 312.461,A -85,B 0,C 180,E1 18579.61,E2 18579.61} C_VEL
LIN {X 0,Y 401.458,Z 312.421,A -85,B 0,C 180,E1 18575.718,E2 18575.718} C_VEL
LIN {X 0,Y 401.461,Z 312.469,A -85,B 0,C 180,E1 18571.869,E2 18571.869} C_VEL
LIN {X 0,Y 401.458,Z 312.467,A -85,B 0,C 180,E1 18567.919,E2 18567.919} C_VEL
LIN {X 0,Y 401.457,Z 312.468,A -85,B 0,C 180,E1 18563.951,E2 18563.951} C_VEL
LIN {X 0,Y 401.459,Z 312.474,A -85,B 0,C 180,E1 18560.102,E2 18560.102} C_VEL
LIN {X 0,Y 401.463,Z 312.479,A -85,B 0,C 180,E1 18556.197,E2 18556.197} C_VEL
LIN {X 0,Y 401.472,Z 312.461,A -85,B 0,C 180,E1 18552.367,E2 18552.367} C_VEL
LIN {X 0,Y 401.48,Z 312.452,A -85,B 0,C 180,E1 18548.449,E2 18548.449} C_VEL
LIN {X 0,Y 401.476,Z 312.469,A -85,B 0,C 180,E1 18544.571,E2 18544.571} C_VEL
LIN {X 0,Y 401.482,Z 312.471,A -85,B 0,C 180,E1 18540.57,E2 18540.57} C_VEL
LIN {X 0,Y 401.462,Z 312.453,A -85,B 0,C 180,E1 18536.536,E2 18536.536} C_VEL
LIN {X 0,Y 401.471,Z 312.459,A -85,B 0,C 180,E1 18532.559,E2 18532.559} C_VEL
LIN {X 0,Y 401.463,Z 312.478,A -85,B 0,C 180,E1 18528.653,E2 18528.653} C_VEL
LIN {X 0,Y 401.448,Z 312.459,A -85,B 0,C 180,E1 18524.84,E2 18524.84} C_VEL
LIN {X 0,Y 401.448,Z 312.46,A -85,B 0,C 180,E1 18520.957,E2 18520.957} C_VEL
LIN {X 0,Y 401.447,Z 312.478,A -85,B 0,C 180,E1 18517.136,E2 18517.136} C_VEL
LIN {X 0,Y 401.451,Z 312.477,A -85,B 0,C 180,E1 18513.205,E2 18513.205} C_VEL
LIN {X 0,Y 401.454,Z 312.472,A -85,B 0,C 180,E1 18509.23,E2 18509.23} C_VEL
LIN {X 0,Y 401.459,Z 312.467,A -85,B 0,C 180,E1 18505.272,E2 18505.272} C_VEL
LIN {X 0,Y 401.469,Z 312.466,A -85,B 0,C 180,E1 18501.444,E2 18501.444} C_VEL
LIN {X 0,Y 401.489,Z 312.466,A -85,B 0,C 180,E1 18497.699,E2 18497.699} C_VEL
LIN {X 0,Y 401.491,Z 312.42,A -85,B 0,C 180,E1 18493.763,E2 18493.763} C_VEL
LIN {X 0,Y 401.525,Z 312.728,A -85,B 0,C 180,E1 18491.528,E2 18491.528} C_VEL
LIN {X 0,Y 402.853,Z 316.073,A -85,B 0,C 180,E1 18490.8,E2 18490.8} C_VEL
LIN {X 0,Y 408.845,Z 330.583,A -85,B 0,C 180,E1 18487.924,E2 18487.924} C_VEL
LIN {X 0,Y 414.239,Z 344.647,A -85,B 0,C 180,E1 18485.449,E2 18485.449} C_VEL
LIN {X 0,Y 426.584,Z 366.634,A -85,B 0,C 180,E1 18483.687,E2 18483.687} C_VEL
LIN {X 0,Y 427.461,Z 371.054,A -85,B 0,C 180,E1 18483.512,E2 18483.512} C_VEL
LIN {X 0,Y 423.636,Z 560.134,A -85,B 0,C 180,E1 18480.345,E2 18480.345} C_VEL
LIN {X 0,Y 422.93,Z 579.467,A -85,B 0,C 180,E1 18479.765,E2 18479.765} C_VEL
LIN {X 0,Y 421.763,Z 597.411,A -85,B 0,C 180,E1 18478.981,E2 18478.981} C_VEL
LIN {X 0,Y 420.184,Z 615,A -85,B 0,C 180,E1 18477.954,E2 18477.954} C_VEL
LIN {X 0,Y 418.23,Z 631.776,A -85,B 0,C 180,E1 18476.708,E2 18476.708} C_VEL
LIN {X 0,Y 416.059,Z 647.549,A -85,B 0,C 180,E1 18475.249,E2 18475.249} C_VEL
LIN {X 0,Y 415.401,Z 651.806,A -85,B 0,C 180,E1 18474.795,E2 18474.795} C_VEL
LIN {X 0,Y 413.589,Z 657.941,A -85,B 0,C 180,E1 18474.181,E2 18474.181} C_VEL
LIN {X 0,Y 406.154,Z 672.262,A -85,B 0,C 180,E1 18472.777,E2 18472.777} C_VEL
LIN {X 0,Y 404.023,Z 677.673,A -85,B 0,C 180,E1 18472.053,E2 18472.053} C_VEL
LIN {X 0,Y 403.855,Z 678.401,A -85,B 0,C 180,E1 18471.937,E2 18471.937} C_VEL
LIN {X 0,Y 401.456,Z 690.73,A -85,B 0,C 180,E1 18469.798,E2 18469.798} C_VEL
LIN {X 0,Y 399.286,Z 701.631,A -85,B 0,C 180,E1 18467.487,E2 18467.487} C_VEL
LIN {X 0,Y 397.364,Z 711.344,A -85,B 0,C 180,E1 18464.931,E2 18464.931} C_VEL
LIN {X 0,Y 395.898,Z 719.007,A -85,B 0,C 180,E1 18462.396,E2 18462.396} C_VEL
LIN {X 0,Y 394.773,Z 725.428,A -85,B 0,C 180,E1 18459.623,E2 18459.623} C_VEL
LIN {X 0,Y 394.021,Z 730.07,A -85,B 0,C 180,E1 18456.85,E2 18456.85} C_VEL
LIN {X 0,Y 393.572,Z 733.178,A -85,B 0,C 180,E1 18453.933,E2 18453.933} C_VEL
LIN {X 0,Y 393.392,Z 734.595,A -85,B 0,C 180,E1 18451.019,E2 18451.019} C_VEL
LIN {X 0,Y 393.423,Z 734.376,A -85,B 0,C 180,E1 18448.107,E2 18448.107} C_VEL
LIN {X 0,Y 393.666,Z 732.51,A -85,B 0,C 180,E1 18445.192,E2 18445.192} C_VEL
LIN {X 0,Y 394.166,Z 729.146,A -85,B 0,C 180,E1 18442.421,E2 18442.421} C_VEL
LIN {X 0,Y 394.99,Z 724.109,A -85,B 0,C 180,E1 18439.647,E2 18439.647} C_VEL
LIN {X 0,Y 396.186,Z 717.445,A -85,B 0,C 180,E1 18436.946,E2 18436.946} C_VEL
LIN {X 0,Y 397.767,Z 709.334,A -85,B 0,C 180,E1 18434.398,E2 18434.398} C_VEL
LIN {X 0,Y 399.711,Z 699.492,A -85,B 0,C 180,E1 18431.931,E2 18431.931} C_VEL
LIN {X 0,Y 401.973,Z 688.118,A -85,B 0,C 180,E1 18429.621,E2 18429.621} C_VEL
LIN {X 0,Y 404.292,Z 676.096,A -85,B 0,C 180,E1 18427.614,E2 18427.614} C_VEL
LIN {X 0,Y 406.707,Z 662.704,A -85,B 0,C 180,E1 18425.761,E2 18425.761} C_VEL
LIN {X 0,Y 409.156,Z 647.802,A -85,B 0,C 180,E1 18424.065,E2 18424.065} C_VEL
LIN {X 0,Y 411.335,Z 632.67,A -85,B 0,C 180,E1 18422.652,E2 18422.652} C_VEL
LIN {X 0,Y 413.382,Z 615.861,A -85,B 0,C 180,E1 18421.387,E2 18421.387} C_VEL
LIN {X 0,Y 415.07,Z 597.887,A -85,B 0,C 180,E1 18420.329,E2 18420.329} C_VEL
LIN {X 0,Y 416.304,Z 579.433,A -85,B 0,C 180,E1 18419.522,E2 18419.522} C_VEL
LIN {X 0,Y 417.013,Z 560.547,A -85,B 0,C 180,E1 18418.955,E2 18418.955} C_VEL
LIN {X 0,Y 420.97,Z 370.964,A -85,B 0,C 180,E1 18415.716,E2 18415.716} C_VEL
LIN {X 0,Y 408.892,Z 349.416,A -85,B 0,C 180,E1 18413.948,E2 18413.948} C_VEL
LIN {X 0,Y 406.12,Z 344.736,A -85,B 0,C 180,E1 18413.498,E2 18413.498} C_VEL
LIN {X 0,Y 400.354,Z 329.96,A -85,B 0,C 180,E1 18410.734,E2 18410.734} C_VEL
LIN {X 0,Y 394.968,Z 317.07,A -85,B 0,C 180,E1 18408.064,E2 18408.064} C_VEL
LIN {X 0,Y 393.56,Z 313.603,A -85,B 0,C 180,E1 18407.242,E2 18407.242} C_VEL
LIN {X 0,Y 393.548,Z 313.459,A -85,B 0,C 180,E1 18403.513,E2 18403.513} C_VEL
LIN {X 0,Y 393.558,Z 313.465,A -85,B 0,C 180,E1 18399.62,E2 18399.62} C_VEL
LIN {X 0,Y 393.554,Z 313.463,A -85,B 0,C 180,E1 18395.614,E2 18395.614} C_VEL
LIN {X 0,Y 393.552,Z 313.464,A -85,B 0,C 180,E1 18391.559,E2 18391.559} C_VEL
LIN {X 0,Y 393.559,Z 313.459,A -85,B 0,C 180,E1 18387.706,E2 18387.706} C_VEL
LIN {X 0,Y 393.556,Z 313.446,A -85,B 0,C 180,E1 18383.667,E2 18383.667} C_VEL
LIN {X 0,Y 393.55,Z 313.44,A -85,B 0,C 180,E1 18379.749,E2 18379.749} C_VEL
LIN {X 0,Y 393.547,Z 313.451,A -85,B 0,C 180,E1 18375.775,E2 18375.775} C_VEL
LIN {X 0,Y 393.531,Z 313.462,A -85,B 0,C 180,E1 18371.877,E2 18371.877} C_VEL
LIN {X 0,Y 393.522,Z 313.442,A -85,B 0,C 180,E1 18367.886,E2 18367.886} C_VEL
LIN {X 0,Y 393.503,Z 313.452,A -85,B 0,C 180,E1 18364.08,E2 18364.08} C_VEL
LIN {X 0,Y 393.488,Z 313.468,A -85,B 0,C 180,E1 18360.291,E2 18360.291} C_VEL
LIN {X 0,Y 393.488,Z 313.45,A -85,B 0,C 180,E1 18356.358,E2 18356.358} C_VEL
LIN {X 0,Y 393.492,Z 313.448,A -85,B 0,C 180,E1 18352.408,E2 18352.408} C_VEL
LIN {X 0,Y 393.501,Z 313.467,A -85,B 0,C 180,E1 18348.42,E2 18348.42} C_VEL
LIN {X 0,Y 393.504,Z 313.467,A -85,B 0,C 180,E1 18344.36,E2 18344.36} C_VEL
LIN {X 0,Y 393.509,Z 313.457,A -85,B 0,C 180,E1 18340.404,E2 18340.404} C_VEL
LIN {X 0,Y 393.516,Z 313.45,A -85,B 0,C 180,E1 18336.49,E2 18336.49} C_VEL
LIN {X 0,Y 393.525,Z 313.449,A -85,B 0,C 180,E1 18332.621,E2 18332.621} C_VEL
LIN {X 0,Y 393.542,Z 313.449,A -85,B 0,C 180,E1 18328.782,E2 18328.782} C_VEL
LIN {X 0,Y 393.549,Z 313.409,A -85,B 0,C 180,E1 18324.891,E2 18324.891} C_VEL
LIN {X 0,Y 393.602,Z 313.683,A -85,B 0,C 180,E1 18321.138,E2 18321.138} C_VEL
LIN {X 0,Y 394.75,Z 316.793,A -85,B 0,C 180,E1 18320.524,E2 18320.524} C_VEL
LIN {X 0,Y 395.956,Z 318.911,A -85,B 0,C 180,E1 18320.104,E2 18320.104} C_VEL
LIN {X 0,Y 401.799,Z 330.761,A -85,B 0,C 180,E1 18317.98,E2 18317.98} C_VEL
LIN {X 0,Y 409.797,Z 348.447,A -85,B 0,C 180,E1 18315.161,E2 18315.161} C_VEL
LIN {X 0,Y 417.495,Z 367.578,A -85,B 0,C 180,E1 18312.471,E2 18312.471} C_VEL
LIN {X 0,Y 419.039,Z 372.186,A -85,B 0,C 180,E1 18311.888,E2 18311.888} C_VEL
LIN {X 0,Y 417.954,Z 382.538,A -85,B 0,C 180,E1 18311.074,E2 18311.074} C_VEL
LIN {X 0,Y 421.871,Z 422.728,A -85,B 0,C 180,E1 18309.787,E2 18309.787} C_VEL
LIN {X 0,Y 415.256,Z 635.275,A -85,B 0,C 180,E1 18305.721,E2 18305.721} C_VEL
LIN {X 0,Y 413.844,Z 656.322,A -85,B 0,C 180,E1 18305.123,E2 18305.123} C_VEL
LIN {X 0,Y 411.921,Z 676.513,A -85,B 0,C 180,E1 18304.314,E2 18304.314} C_VEL
LIN {X 0,Y 409.615,Z 696.882,A -85,B 0,C 180,E1 18303.229,E2 18303.229} C_VEL
LIN {X 0,Y 407.252,Z 715.888,A -85,B 0,C 180,E1 18301.942,E2 18301.942} C_VEL
LIN {X 0,Y 404.765,Z 734.249,A -85,B 0,C 180,E1 18300.423,E2 18300.423} C_VEL
LIN {X 0,Y 402.21,Z 752.538,A -85,B 0,C 180,E1 18298.589,E2 18298.589} C_VEL
LIN {X 0,Y 399.787,Z 769.779,A -85,B 0,C 180,E1 18296.514,E2 18296.514} C_VEL
LIN {X 0,Y 397.601,Z 785.904,A -85,B 0,C 180,E1 18294.198,E2 18294.198} C_VEL
LIN {X 0,Y 395.835,Z 799.983,A -85,B 0,C 180,E1 18291.796,E2 18291.796} C_VEL
LIN {X 0,Y 394.463,Z 812.649,A -85,B 0,C 180,E1 18289.239,E2 18289.239} C_VEL
LIN {X 0,Y 393.476,Z 823.859,A -85,B 0,C 180,E1 18286.535,E2 18286.535} C_VEL
LIN {X 0,Y 392.863,Z 833.534,A -85,B 0,C 180,E1 18283.691,E2 18283.691} C_VEL
LIN {X 0,Y 392.593,Z 841.224,A -85,B 0,C 180,E1 18280.863,E2 18280.863} C_VEL
LIN {X 0,Y 392.532,Z 847.083,A -85,B 0,C 180,E1 18278.053,E2 18278.053} C_VEL
LIN {X 0,Y 392.606,Z 851.096,A -85,B 0,C 180,E1 18275.26,E2 18275.26} C_VEL
LIN {X 0,Y 392.687,Z 853.424,A -85,B 0,C 180,E1 18272.481,E2 18272.481} C_VEL
LIN {X 0,Y 392.717,Z 854.138,A -85,B 0,C 180,E1 18269.854,E2 18269.854} C_VEL
LIN {X 0,Y 392.683,Z 853.267,A -85,B 0,C 180,E1 18267.227,E2 18267.227} C_VEL
LIN {X 0,Y 392.601,Z 850.733,A -85,B 0,C 180,E1 18264.447,E2 18264.447} C_VEL
LIN {X 0,Y 392.534,Z 846.526,A -85,B 0,C 180,E1 18261.652,E2 18261.652} C_VEL
LIN {X 0,Y 392.597,Z 840.885,A -85,B 0,C 180,E1 18258.989,E2 18258.989} C_VEL
LIN {X 0,Y 392.864,Z 833.534,A -85,B 0,C 180,E1 18256.309,E2 18256.309} C_VEL
LIN {X 0,Y 393.477,Z 823.854,A -85,B 0,C 180,E1 18253.465,E2 18253.465} C_VEL
LIN {X 0,Y 394.464,Z 812.641,A -85,B 0,C 180,E1 18250.761,E2 18250.761} C_VEL
LIN {X 0,Y 395.833,Z 799.971,A -85,B 0,C 180,E1 18248.204,E2 18248.204} C_VEL
LIN {X 0,Y 397.6,Z 785.884,A -85,B 0,C 180,E1 18245.802,E2 18245.802} C_VEL
LIN {X 0,Y 399.785,Z 769.75,A -85,B 0,C 180,E1 18243.486,E2 18243.486} C_VEL
LIN {X 0,Y 402.303,Z 751.833,A -85,B 0,C 180,E1 18241.337,E2 18241.337} C_VEL
LIN {X 0,Y 404.863,Z 733.507,A -85,B 0,C 180,E1 18239.511,E2 18239.511} C_VEL
LIN {X 0,Y 407.504,Z 713.952,A -85,B 0,C 180,E1 18237.914,E2 18237.914} C_VEL
LIN {X 0,Y 409.943,Z 694.091,A -85,B 0,C 180,E1 18236.607,E2 18236.607} C_VEL
LIN {X 0,Y 412.077,Z 674.905,A -85,B 0,C 180,E1 18235.617,E2 18235.617} C_VEL
LIN {X 0,Y 414.012,Z 653.942,A -85,B 0,C 180,E1 18234.802,E2 18234.802} C_VEL
LIN {X 0,Y 415.363,Z 632.112,A -85,B 0,C 180,E1 18234.215,E2 18234.215} C_VEL
LIN {X 0,Y 421.873,Z 421.052,A -85,B 0,C 180,E1 18230.186,E2 18230.186} C_VEL
LIN {X 0,Y 417.909,Z 381.477,A -85,B 0,C 180,E1 18228.879,E2 18228.879} C_VEL
LIN {X 0,Y 419.038,Z 371.813,A -85,B 0,C 180,E1 18228.081,E2 18228.081} C_VEL
LIN {X 0,Y 411.753,Z 353.239,A -85,B 0,C 180,E1 18225.554,E2 18225.554} C_VEL
LIN {X 0,Y 404.51,Z 336.713,A -85,B 0,C 180,E1 18223.016,E2 18223.016} C_VEL
LIN {X 0,Y 397.474,Z 321.825,A -85,B 0,C 180,E1 18220.466,E2 18220.466} C_VEL
LIN {X 0,Y 393.692,Z 314.172,A -85,B 0,C 180,E1 18219.033,E2 18219.033} C_VEL
LIN {X 0,Y 393.562,Z 313.469,A -85,B 0,C 180,E1 18218.68,E2 18218.68} C_VEL
LIN {X 0,Y 393.552,Z 313.417,A -85,B 0,C 180,E1 18214.687,E2 18214.687} C_VEL
LIN {X 0,Y 393.565,Z 313.448,A -85,B 0,C 180,E1 18210.706,E2 18210.706} C_VEL
LIN {X 0,Y 393.558,Z 313.448,A -85,B 0,C 180,E1 18206.723,E2 18206.723} C_VEL
LIN {X 0,Y 393.565,Z 313.444,A -85,B 0,C 180,E1 18202.715,E2 18202.715} C_VEL
LIN {X 0,Y 393.55,Z 313.443,A -85,B 0,C 180,E1 18198.67,E2 18198.67} C_VEL
LIN {X 0,Y 393.554,Z 313.448,A -85,B 0,C 180,E1 18194.717,E2 18194.717} C_VEL
LIN {X 0,Y 393.541,Z 313.466,A -85,B 0,C 180,E1 18190.688,E2 18190.688} C_VEL
LIN {X 0,Y 393.548,Z 313.454,A -85,B 0,C 180,E1 18186.608,E2 18186.608} C_VEL
LIN {X 0,Y 393.531,Z 313.44,A -85,B 0,C 180,E1 18182.621,E2 18182.621} C_VEL
LIN {X 0,Y 393.522,Z 313.456,A -85,B 0,C 180,E1 18178.689,E2 18178.689} C_VEL
LIN {X 0,Y 393.515,Z 313.464,A -85,B 0,C 180,E1 18174.751,E2 18174.751} C_VEL
LIN {X 0,Y 393.501,Z 313.442,A -85,B 0,C 180,E1 18170.936,E2 18170.936} C_VEL
LIN {X 0,Y 393.499,Z 313.457,A -85,B 0,C 180,E1 18167.079,E2 18167.079} C_VEL
LIN {X 0,Y 393.502,Z 313.467,A -85,B 0,C 180,E1 18163.162,E2 18163.162} C_VEL
LIN {X 0,Y 393.505,Z 313.455,A -85,B 0,C 180,E1 18159.162,E2 18159.162} C_VEL
LIN {X 0,Y 393.507,Z 313.444,A -85,B 0,C 180,E1 18155.213,E2 18155.213} C_VEL
LIN {X 0,Y 393.513,Z 313.453,A -85,B 0,C 180,E1 18151.231,E2 18151.231} C_VEL
LIN {X 0,Y 393.518,Z 313.46,A -85,B 0,C 180,E1 18147.235,E2 18147.235} C_VEL
LIN {X 0,Y 393.524,Z 313.464,A -85,B 0,C 180,E1 18143.338,E2 18143.338} C_VEL
LIN {X 0,Y 393.535,Z 313.458,A -85,B 0,C 180,E1 18139.426,E2 18139.426} C_VEL
LIN {X 0,Y 393.538,Z 313.431,A -85,B 0,C 180,E1 18135.474,E2 18135.474} C_VEL
LIN {X 0,Y 393.567,Z 313.66,A -85,B 0,C 180,E1 18132.613,E2 18132.613} C_VEL
LIN {X 0,Y 398.812,Z 326.272,A -85,B 0,C 180,E1 18129.899,E2 18129.899} C_VEL
LIN {X 0,Y 404.332,Z 340.049,A -85,B 0,C 180,E1 18127.225,E2 18127.225} C_VEL
LIN {X 0,Y 406.421,Z 345.401,A -85,B 0,C 180,E1 18126.322,E2 18126.322} C_VEL
LIN {X 0,Y 417.747,Z 365.108,A -85,B 0,C 180,E1 18124.638,E2 18124.638} C_VEL
LIN {X 0,Y 421.06,Z 371.655,A -85,B 0,C 180,E1 18124.156,E2 18124.156} C_VEL
LIN {X 0,Y 416.97,Z 560.855,A -85,B 0,C 180,E1 18120.941,E2 18120.941} C_VEL
LIN {X 0,Y 416.238,Z 580.043,A -85,B 0,C 180,E1 18120.36,E2 18120.36} C_VEL
LIN {X 0,Y 414.951,Z 598.933,A -85,B 0,C 180,E1 18119.521,E2 18119.521} C_VEL
LIN {X 0,Y 413.27,Z 616.635,A -85,B 0,C 180,E1 18118.464,E2 18118.464} C_VEL
LIN {X 0,Y 411.226,Z 633.289,A -85,B 0,C 180,E1 18117.2,E2 18117.2} C_VEL
LIN {X 0,Y 408.847,Z 649.658,A -85,B 0,C 180,E1 18115.649,E2 18115.649} C_VEL
LIN {X 0,Y 406.337,Z 664.754,A -85,B 0,C 180,E1 18113.884,E2 18113.884} C_VEL
LIN {X 0,Y 403.855,Z 678.401,A -85,B 0,C 180,E1 18111.937,E2 18111.937} C_VEL
LIN {X 0,Y 401.943,Z 683.676,A -85,B 0,C 180,E1 18111.153,E2 18111.153} C_VEL
LIN {X 0,Y 393.99,Z 696.367,A -85,B 0,C 180,E1 18109.222,E2 18109.222} C_VEL
LIN {X 0,Y 392.177,Z 700.714,A -85,B 0,C 180,E1 18108.337,E2 18108.337} C_VEL
LIN {X 0,Y 390.193,Z 710.225,A -85,B 0,C 180,E1 18105.913,E2 18105.913} C_VEL
LIN {X 0,Y 388.465,Z 718.608,A -85,B 0,C 180,E1 18103.242,E2 18103.242} C_VEL
LIN {X 0,Y 387.22,Z 725.118,A -85,B 0,C 180,E1 18100.564,E2 18100.564} C_VEL
LIN {X 0,Y 386.334,Z 730.204,A -85,B 0,C 180,E1 18097.734,E2 18097.734} C_VEL
LIN {X 0,Y 385.788,Z 733.618,A -85,B 0,C 180,E1 18094.906,E2 18094.906} C_VEL
LIN {X 0,Y 385.519,Z 735.537,A -85,B 0,C 180,E1 18091.932,E2 18091.932} C_VEL
LIN {X 0,Y 385.481,Z 735.811,A -85,B 0,C 180,E1 18088.96,E2 18088.96} C_VEL
LIN {X 0,Y 385.669,Z 734.451,A -85,B 0,C 180,E1 18085.986,E2 18085.986} C_VEL
LIN {X 0,Y 386.108,Z 731.587,A -85,B 0,C 180,E1 18083.159,E2 18083.159} C_VEL
LIN {X 0,Y 386.879,Z 727.097,A -85,B 0,C 180,E1 18080.329,E2 18080.329} C_VEL
LIN {X 0,Y 388.037,Z 720.843,A -85,B 0,C 180,E1 18077.5,E2 18077.5} C_VEL
LIN {X 0,Y 389.611,Z 713.082,A -85,B 0,C 180,E1 18074.826,E2 18074.826} C_VEL
LIN {X 0,Y 391.536,Z 703.858,A -85,B 0,C 180,E1 18072.309,E2 18072.309} C_VEL
LIN {X 0,Y 393.775,Z 693.191,A -85,B 0,C 180,E1 18069.954,E2 18069.954} C_VEL
LIN {X 0,Y 396.276,Z 681.051,A -85,B 0,C 180,E1 18067.762,E2 18067.762} C_VEL
LIN {X 0,Y 398.813,Z 667.874,A -85,B 0,C 180,E1 18065.802,E2 18065.802} C_VEL
LIN {X 0,Y 401.423,Z 653.145,A -85,B 0,C 180,E1 18064,E2 18064} C_VEL
LIN {X 0,Y 403.781,Z 638.127,A -85,B 0,C 180,E1 18062.496,E2 18062.496} C_VEL
LIN {X 0,Y 406.017,Z 621.425,A -85,B 0,C 180,E1 18061.141,E2 18061.141} C_VEL
LIN {X 0,Y 407.797,Z 604.816,A -85,B 0,C 180,E1 18060.07,E2 18060.07} C_VEL
LIN {X 0,Y 409.272,Z 586.2,A -85,B 0,C 180,E1 18059.155,E2 18059.155} C_VEL
LIN {X 0,Y 410.213,Z 566.946,A -85,B 0,C 180,E1 18058.489,E2 18058.489} C_VEL
LIN {X 0,Y 410.706,Z 542.868,A -85,B 0,C 180,E1 18057.988,E2 18057.988} C_VEL
LIN {X 0,Y 414.637,Z 373.964,A -85,B 0,C 180,E1 18055.1,E2 18055.1} C_VEL
LIN {X 0,Y 403.294,Z 353.738,A -85,B 0,C 180,E1 18053.385,E2 18053.385} C_VEL
LIN {X 0,Y 398.148,Z 345.046,A -85,B 0,C 180,E1 18052.52,E2 18052.52} C_VEL
LIN {X 0,Y 391.902,Z 329.245,A -85,B 0,C 180,E1 18049.416,E2 18049.416} C_VEL
LIN {X 0,Y 387.041,Z 318.11,A -85,B 0,C 180,E1 18046.978,E2 18046.978} C_VEL
LIN {X 0,Y 385.647,Z 314.605,A -85,B 0,C 180,E1 18046.118,E2 18046.118} C_VEL
LIN {X 0,Y 385.622,Z 314.44,A -85,B 0,C 180,E1 18042.138,E2 18042.138} C_VEL
LIN {X 0,Y 385.621,Z 314.435,A -85,B 0,C 180,E1 18038.105,E2 18038.105} C_VEL
LIN {X 0,Y 385.615,Z 314.434,A -85,B 0,C 180,E1 18034.061,E2 18034.061} C_VEL
LIN {X 0,Y 385.617,Z 314.433,A -85,B 0,C 180,E1 18030.003,E2 18030.003} C_VEL
LIN {X 0,Y 385.599,Z 314.444,A -85,B 0,C 180,E1 18026.156,E2 18026.156} C_VEL
LIN {X 0,Y 385.588,Z 314.455,A -85,B 0,C 180,E1 18022.226,E2 18022.226} C_VEL
LIN {X 0,Y 385.578,Z 314.444,A -85,B 0,C 180,E1 18018.287,E2 18018.287} C_VEL
LIN {X 0,Y 385.566,Z 314.43,A -85,B 0,C 180,E1 18014.416,E2 18014.416} C_VEL
LIN {X 0,Y 385.563,Z 314.453,A -85,B 0,C 180,E1 18010.459,E2 18010.459} C_VEL
LIN {X 0,Y 385.555,Z 314.456,A -85,B 0,C 180,E1 18006.552,E2 18006.552} C_VEL
LIN {X 0,Y 385.548,Z 314.432,A -85,B 0,C 180,E1 18002.527,E2 18002.527} C_VEL
LIN {X 0,Y 385.547,Z 314.444,A -85,B 0,C 180,E1 17998.514,E2 17998.514} C_VEL
LIN {X 0,Y 385.554,Z 314.456,A -85,B 0,C 180,E1 17994.494,E2 17994.494} C_VEL
LIN {X 0,Y 385.558,Z 314.445,A -85,B 0,C 180,E1 17990.447,E2 17990.447} C_VEL
LIN {X 0,Y 385.561,Z 314.432,A -85,B 0,C 180,E1 17986.351,E2 17986.351} C_VEL
LIN {X 0,Y 385.566,Z 314.441,A -85,B 0,C 180,E1 17982.338,E2 17982.338} C_VEL
LIN {X 0,Y 385.572,Z 314.449,A -85,B 0,C 180,E1 17978.234,E2 17978.234} C_VEL
LIN {X 0,Y 385.579,Z 314.451,A -85,B 0,C 180,E1 17974.131,E2 17974.131} C_VEL
LIN {X 0,Y 385.58,Z 314.45,A -85,B 0,C 180,E1 17970.14,E2 17970.14} C_VEL
LIN {X 0,Y 385.581,Z 314.427,A -85,B 0,C 180,E1 17966.076,E2 17966.076} C_VEL
LIN {X 0,Y 385.606,Z 314.558,A -85,B 0,C 180,E1 17962.365,E2 17962.365} C_VEL
LIN {X 0,Y 386.069,Z 316.334,A -85,B 0,C 180,E1 17961.948,E2 17961.948} C_VEL
LIN {X 0,Y 387.999,Z 319.736,A -85,B 0,C 180,E1 17961.23,E2 17961.23} C_VEL
LIN {X 0,Y 394.474,Z 332.948,A -85,B 0,C 180,E1 17958.776,E2 17958.776} C_VEL
LIN {X 0,Y 402.152,Z 349.684,A -85,B 0,C 180,E1 17955.98,E2 17955.98} C_VEL
LIN {X 0,Y 409.948,Z 368.876,A -85,B 0,C 180,E1 17953.176,E2 17953.176} C_VEL
LIN {X 0,Y 412.124,Z 375.317,A -85,B 0,C 180,E1 17952.316,E2 17952.316} C_VEL
LIN {X 0,Y 411.447,Z 382.221,A -85,B 0,C 180,E1 17951.784,E2 17951.784} C_VEL
LIN {X 0,Y 415.419,Z 423.705,A -85,B 0,C 180,E1 17950.425,E2 17950.425} C_VEL
LIN {X 0,Y 408.519,Z 634.944,A -85,B 0,C 180,E1 17946.328,E2 17946.328} C_VEL
LIN {X 0,Y 407.039,Z 655.856,A -85,B 0,C 180,E1 17945.721,E2 17945.721} C_VEL
LIN {X 0,Y 405.023,Z 676.041,A -85,B 0,C 180,E1 17944.896,E2 17944.896} C_VEL
LIN {X 0,Y 402.603,Z 696.28,A -85,B 0,C 180,E1 17943.799,E2 17943.799} C_VEL
LIN {X 0,Y 399.99,Z 716.125,A -85,B 0,C 180,E1 17942.423,E2 17942.423} C_VEL
LIN {X 0,Y 397.388,Z 734.247,A -85,B 0,C 180,E1 17940.881,E2 17940.881} C_VEL
LIN {X 0,Y 394.81,Z 751.702,A -85,B 0,C 180,E1 17939.093,E2 17939.093} C_VEL
LIN {X 0,Y 392.246,Z 768.898,A -85,B 0,C 180,E1 17936.982,E2 17936.982} C_VEL
LIN {X 0,Y 389.928,Z 784.982,A -85,B 0,C 180,E1 17934.625,E2 17934.625} C_VEL
LIN {X 0,Y 388.003,Z 799.438,A -85,B 0,C 180,E1 17932.1,E2 17932.1} C_VEL
LIN {X 0,Y 386.562,Z 811.997,A -85,B 0,C 180,E1 17929.491,E2 17929.491} C_VEL
LIN {X 0,Y 385.527,Z 823.11,A -85,B 0,C 180,E1 17926.73,E2 17926.73} C_VEL
LIN {X 0,Y 384.897,Z 832.698,A -85,B 0,C 180,E1 17923.827,E2 17923.827} C_VEL
LIN {X 0,Y 384.626,Z 840.306,A -85,B 0,C 180,E1 17920.939,E2 17920.939} C_VEL
LIN {X 0,Y 384.583,Z 845.847,A -85,B 0,C 180,E1 17918.221,E2 17918.221} C_VEL
LIN {X 0,Y 384.675,Z 849.795,A -85,B 0,C 180,E1 17915.437,E2 17915.437} C_VEL
LIN {X 0,Y 384.771,Z 852.141,A -85,B 0,C 180,E1 17912.681,E2 17912.681} C_VEL
LIN {X 0,Y 384.812,Z 852.954,A -85,B 0,C 180,E1 17910,E2 17910} C_VEL
LIN {X 0,Y 384.772,Z 852.14,A -85,B 0,C 180,E1 17907.319,E2 17907.319} C_VEL
LIN {X 0,Y 384.673,Z 849.694,A -85,B 0,C 180,E1 17904.481,E2 17904.481} C_VEL
LIN {X 0,Y 384.583,Z 845.846,A -85,B 0,C 180,E1 17901.779,E2 17901.779} C_VEL
LIN {X 0,Y 384.632,Z 839.966,A -85,B 0,C 180,E1 17898.909,E2 17898.909} C_VEL
LIN {X 0,Y 384.897,Z 832.697,A -85,B 0,C 180,E1 17896.173,E2 17896.173} C_VEL
LIN {X 0,Y 385.527,Z 823.103,A -85,B 0,C 180,E1 17893.27,E2 17893.27} C_VEL
LIN {X 0,Y 386.562,Z 811.985,A -85,B 0,C 180,E1 17890.509,E2 17890.509} C_VEL
LIN {X 0,Y 388.003,Z 799.422,A -85,B 0,C 180,E1 17887.9,E2 17887.9} C_VEL
LIN {X 0,Y 389.927,Z 784.958,A -85,B 0,C 180,E1 17885.375,E2 17885.375} C_VEL
LIN {X 0,Y 392.244,Z 768.864,A -85,B 0,C 180,E1 17883.017,E2 17883.017} C_VEL
LIN {X 0,Y 394.897,Z 751.073,A -85,B 0,C 180,E1 17880.839,E2 17880.839} C_VEL
LIN {X 0,Y 397.624,Z 732.652,A -85,B 0,C 180,E1 17878.971,E2 17878.971} C_VEL
LIN {X 0,Y 400.293,Z 713.881,A -85,B 0,C 180,E1 17877.407,E2 17877.407} C_VEL
LIN {X 0,Y 402.784,Z 694.725,A -85,B 0,C 180,E1 17876.111,E2 17876.111} C_VEL
LIN {X 0,Y 405.099,Z 675.163,A -85,B 0,C 180,E1 17875.068,E2 17875.068} C_VEL
LIN {X 0,Y 407.181,Z 653.862,A -85,B 0,C 180,E1 17874.217,E2 17874.217} C_VEL
LIN {X 0,Y 408.624,Z 631.863,A -85,B 0,C 180,E1 17873.61,E2 17873.61} C_VEL
LIN {X 0,Y 415.42,Z 422.205,A -85,B 0,C 180,E1 17869.553,E2 17869.553} C_VEL
LIN {X 0,Y 411.396,Z 380.893,A -85,B 0,C 180,E1 17868.154,E2 17868.154} C_VEL
LIN {X 0,Y 412.119,Z 374.753,A -85,B 0,C 180,E1 17867.625,E2 17867.625} C_VEL
LIN {X 0,Y 404.692,Z 355.738,A -85,B 0,C 180,E1 17864.959,E2 17864.959} C_VEL
LIN {X 0,Y 397.175,Z 338.608,A -85,B 0,C 180,E1 17862.233,E2 17862.233} C_VEL
LIN {X 0,Y 389.71,Z 323.102,A -85,B 0,C 180,E1 17859.445,E2 17859.445} C_VEL
LIN {X 0,Y 387.178,Z 318.289,A -85,B 0,C 180,E1 17858.489,E2 17858.489} C_VEL
LIN {X 0,Y 385.625,Z 314.681,A -85,B 0,C 180,E1 17857.727,E2 17857.727} C_VEL
LIN {X 0,Y 385.601,Z 314.41,A -85,B 0,C 180,E1 17854.458,E2 17854.458} C_VEL
LIN {X 0,Y 385.614,Z 314.439,A -85,B 0,C 180,E1 17850.544,E2 17850.544} C_VEL
LIN {X 0,Y 385.611,Z 314.438,A -85,B 0,C 180,E1 17846.552,E2 17846.552} C_VEL
LIN {X 0,Y 385.614,Z 314.434,A -85,B 0,C 180,E1 17842.566,E2 17842.566} C_VEL
LIN {X 0,Y 385.609,Z 314.431,A -85,B 0,C 180,E1 17838.598,E2 17838.598} C_VEL
LIN {X 0,Y 385.615,Z 314.434,A -85,B 0,C 180,E1 17834.567,E2 17834.567} C_VEL
LIN {X 0,Y 385.6,Z 314.451,A -85,B 0,C 180,E1 17830.457,E2 17830.457} C_VEL
LIN {X 0,Y 385.6,Z 314.446,A -85,B 0,C 180,E1 17826.401,E2 17826.401} C_VEL
LIN {X 0,Y 385.589,Z 314.429,A -85,B 0,C 180,E1 17822.378,E2 17822.378} C_VEL
LIN {X 0,Y 385.593,Z 314.44,A -85,B 0,C 180,E1 17818.514,E2 17818.514} C_VEL
LIN {X 0,Y 385.594,Z 314.456,A -85,B 0,C 180,E1 17814.345,E2 17814.345} C_VEL
LIN {X 0,Y 385.592,Z 314.431,A -85,B 0,C 180,E1 17810.447,E2 17810.447} C_VEL
LIN {X 0,Y 385.607,Z 314.428,A -85,B 0,C 180,E1 17806.352,E2 17806.352} C_VEL
LIN {X 0,Y 385.607,Z 314.448,A -85,B 0,C 180,E1 17802.339,E2 17802.339} C_VEL
LIN {X 0,Y 385.621,Z 314.448,A -85,B 0,C 180,E1 17798.236,E2 17798.236} C_VEL
LIN {X 0,Y 385.611,Z 314.436,A -85,B 0,C 180,E1 17794.121,E2 17794.121} C_VEL
LIN {X 0,Y 385.629,Z 314.431,A -85,B 0,C 180,E1 17790.144,E2 17790.144} C_VEL
LIN {X 0,Y 385.618,Z 314.434,A -85,B 0,C 180,E1 17786.067,E2 17786.067} C_VEL
LIN {X 0,Y 385.625,Z 314.435,A -85,B 0,C 180,E1 17782.017,E2 17782.017} C_VEL
LIN {X 0,Y 385.624,Z 314.438,A -85,B 0,C 180,E1 17778.013,E2 17778.013} C_VEL
LIN {X 0,Y 385.626,Z 314.47,A -85,B 0,C 180,E1 17773.879,E2 17773.879} C_VEL
LIN {X 0,Y 385.859,Z 315.653,A -85,B 0,C 180,E1 17773.485,E2 17773.485} C_VEL
LIN {X 0,Y 389.443,Z 323.771,A -85,B 0,C 180,E1 17771.658,E2 17771.658} C_VEL
LIN {X 0,Y 394.691,Z 336.105,A -85,B 0,C 180,E1 17769.075,E2 17769.075} C_VEL
LIN {X 0,Y 398.547,Z 345.9,A -85,B 0,C 180,E1 17767.259,E2 17767.259} C_VEL
LIN {X 0,Y 410.134,Z 365.728,A -85,B 0,C 180,E1 17765.461,E2 17765.461} C_VEL
LIN {X 0,Y 414.661,Z 374.464,A -85,B 0,C 180,E1 17764.781,E2 17764.781} C_VEL
LIN {X 0,Y 410.35,Z 561.559,A -85,B 0,C 180,E1 17761.555,E2 17761.555} C_VEL
LIN {X 0,Y 409.587,Z 580.645,A -85,B 0,C 180,E1 17760.971,E2 17760.971} C_VEL
LIN {X 0,Y 408.262,Z 599.362,A -85,B 0,C 180,E1 17760.135,E2 17760.135} C_VEL
LIN {X 0,Y 406.502,Z 617.193,A -85,B 0,C 180,E1 17759.063,E2 17759.063} C_VEL
LIN {X 0,Y 404.361,Z 633.932,A -85,B 0,C 180,E1 17757.781,E2 17757.781} C_VEL
LIN {X 0,Y 401.982,Z 649.691,A -85,B 0,C 180,E1 17756.278,E2 17756.278} C_VEL
LIN {X 0,Y 399.332,Z 665.051,A -85,B 0,C 180,E1 17754.48,E2 17754.48} C_VEL
LIN {X 0,Y 396.734,Z 678.706,A -85,B 0,C 180,E1 17752.524,E2 17752.524} C_VEL
LIN {X 0,Y 394.177,Z 691.263,A -85,B 0,C 180,E1 17750.335,E2 17750.335} C_VEL
LIN {X 0,Y 392.177,Z 700.714,A -85,B 0,C 180,E1 17748.337,E2 17748.337} C_VEL
LIN {X 0,Y 390.401,Z 704.945,A -85,B 0,C 180,E1 17747.419,E2 17747.419} C_VEL
LIN {X 0,Y 383.096,Z 714.504,A -85,B 0,C 180,E1 17745.235,E2 17745.235} C_VEL
LIN {X 0,Y 381.201,Z 717.867,A -85,B 0,C 180,E1 17744.223,E2 17744.223} C_VEL
LIN {X 0,Y 381.081,Z 718.294,A -85,B 0,C 180,E1 17744.07,E2 17744.07} C_VEL
LIN {X 0,Y 379.62,Z 725.372,A -85,B 0,C 180,E1 17741.239,E2 17741.239} C_VEL
LIN {X 0,Y 378.609,Z 730.728,A -85,B 0,C 180,E1 17738.351,E2 17738.351} C_VEL
LIN {X 0,Y 377.947,Z 734.538,A -85,B 0,C 180,E1 17735.313,E2 17735.313} C_VEL
LIN {X 0,Y 377.628,Z 736.618,A -85,B 0,C 180,E1 17732.276,E2 17732.276} C_VEL
LIN {X 0,Y 377.569,Z 737.051,A -85,B 0,C 180,E1 17729.241,E2 17729.241} C_VEL
LIN {X 0,Y 377.738,Z 735.857,A -85,B 0,C 180,E1 17726.206,E2 17726.206} C_VEL
LIN {X 0,Y 378.21,Z 732.98,A -85,B 0,C 180,E1 17723.168,E2 17723.168} C_VEL
LIN {X 0,Y 379.011,Z 728.584,A -85,B 0,C 180,E1 17720.28,E2 17720.28} C_VEL
LIN {X 0,Y 380.217,Z 722.434,A -85,B 0,C 180,E1 17717.393,E2 17717.393} C_VEL
LIN {X 0,Y 381.855,Z 714.787,A -85,B 0,C 180,E1 17714.666,E2 17714.666} C_VEL
LIN {X 0,Y 383.859,Z 705.693,A -85,B 0,C 180,E1 17712.1,E2 17712.1} C_VEL
LIN {X 0,Y 386.186,Z 695.176,A -85,B 0,C 180,E1 17709.701,E2 17709.701} C_VEL
LIN {X 0,Y 388.781,Z 683.214,A -85,B 0,C 180,E1 17707.469,E2 17707.469} C_VEL
LIN {X 0,Y 391.557,Z 669.548,A -85,B 0,C 180,E1 17705.377,E2 17705.377} C_VEL
LIN {X 0,Y 394.32,Z 654.709,A -85,B 0,C 180,E1 17703.52,E2 17703.52} C_VEL
LIN {X 0,Y 396.938,Z 638.786,A -85,B 0,C 180,E1 17701.899,E2 17701.899} C_VEL
LIN {X 0,Y 399.22,Z 622.45,A -85,B 0,C 180,E1 17700.558,E2 17700.558} C_VEL
LIN {X 0,Y 401.139,Z 605.268,A -85,B 0,C 180,E1 17699.438,E2 17699.438} C_VEL
LIN {X 0,Y 402.681,Z 586.474,A -85,B 0,C 180,E1 17698.51,E2 17698.51} C_VEL
LIN {X 0,Y 403.641,Z 567.558,A -85,B 0,C 180,E1 17697.853,E2 17697.853} C_VEL
LIN {X 0,Y 404.166,Z 543.341,A -85,B 0,C 180,E1 17697.344,E2 17697.344} C_VEL
LIN {X 0,Y 408.292,Z 376.865,A -85,B 0,C 180,E1 17694.457,E2 17694.457} C_VEL
LIN {X 0,Y 397.395,Z 357.5,A -85,B 0,C 180,E1 17692.751,E2 17692.751} C_VEL
LIN {X 0,Y 390.285,Z 345.742,A -85,B 0,C 180,E1 17691.54,E2 17691.54} C_VEL
LIN {X 0,Y 384.365,Z 330.944,A -85,B 0,C 180,E1 17688.52,E2 17688.52} C_VEL
LIN {X 0,Y 379.18,Z 319.159,A -85,B 0,C 180,E1 17685.827,E2 17685.827} C_VEL
LIN {X 0,Y 377.685,Z 315.625,A -85,B 0,C 180,E1 17684.919,E2 17684.919} C_VEL
LIN {X 0,Y 377.652,Z 315.43,A -85,B 0,C 180,E1 17681.015,E2 17681.015} C_VEL
LIN {X 0,Y 377.648,Z 315.433,A -85,B 0,C 180,E1 17676.913,E2 17676.913} C_VEL
LIN {X 0,Y 377.644,Z 315.432,A -85,B 0,C 180,E1 17672.872,E2 17672.872} C_VEL
LIN {X 0,Y 377.64,Z 315.427,A -85,B 0,C 180,E1 17668.795,E2 17668.795} C_VEL
LIN {X 0,Y 377.636,Z 315.42,A -85,B 0,C 180,E1 17664.73,E2 17664.73} C_VEL
LIN {X 0,Y 377.634,Z 315.428,A -85,B 0,C 180,E1 17660.619,E2 17660.619} C_VEL
LIN {X 0,Y 377.63,Z 315.444,A -85,B 0,C 180,E1 17656.575,E2 17656.575} C_VEL
LIN {X 0,Y 377.623,Z 315.438,A -85,B 0,C 180,E1 17652.54,E2 17652.54} C_VEL
LIN {X 0,Y 377.616,Z 315.417,A -85,B 0,C 180,E1 17648.527,E2 17648.527} C_VEL
LIN {X 0,Y 377.614,Z 315.439,A -85,B 0,C 180,E1 17644.556,E2 17644.556} C_VEL
LIN {X 0,Y 377.61,Z 315.445,A -85,B 0,C 180,E1 17640.455,E2 17640.455} C_VEL
LIN {X 0,Y 377.611,Z 315.425,A -85,B 0,C 180,E1 17636.357,E2 17636.357} C_VEL
LIN {X 0,Y 377.615,Z 315.423,A -85,B 0,C 180,E1 17632.393,E2 17632.393} C_VEL
LIN {X 0,Y 377.623,Z 315.445,A -85,B 0,C 180,E1 17628.391,E2 17628.391} C_VEL
LIN {X 0,Y 377.627,Z 315.445,A -85,B 0,C 180,E1 17624.332,E2 17624.332} C_VEL
LIN {X 0,Y 377.632,Z 315.437,A -85,B 0,C 180,E1 17620.19,E2 17620.19} C_VEL
LIN {X 0,Y 377.636,Z 315.43,A -85,B 0,C 180,E1 17616.103,E2 17616.103} C_VEL
LIN {X 0,Y 377.641,Z 315.43,A -85,B 0,C 180,E1 17612.055,E2 17612.055} C_VEL
LIN {X 0,Y 377.646,Z 315.434,A -85,B 0,C 180,E1 17608.027,E2 17608.027} C_VEL
LIN {X 0,Y 377.641,Z 315.379,A -85,B 0,C 180,E1 17604.001,E2 17604.001} C_VEL
LIN {X 0,Y 377.755,Z 315.934,A -85,B 0,C 180,E1 17603.449,E2 17603.449} C_VEL
LIN {X 0,Y 379.388,Z 319.449,A -85,B 0,C 180,E1 17602.688,E2 17602.688} C_VEL
LIN {X 0,Y 384.547,Z 329.646,A -85,B 0,C 180,E1 17600.623,E2 17600.623} C_VEL
LIN {X 0,Y 391.456,Z 344.031,A -85,B 0,C 180,E1 17597.995,E2 17597.995} C_VEL
LIN {X 0,Y 398.852,Z 361.24,A -85,B 0,C 180,E1 17595.218,E2 17595.218} C_VEL
LIN {X 0,Y 405.282,Z 378.055,A -85,B 0,C 180,E1 17592.793,E2 17592.793} C_VEL
LIN {X 0,Y 404.997,Z 381.83,A -85,B 0,C 180,E1 17592.52,E2 17592.52} C_VEL
LIN {X 0,Y 409.019,Z 424.703,A -85,B 0,C 180,E1 17591.082,E2 17591.082} C_VEL
LIN {X 0,Y 401.833,Z 634.597,A -85,B 0,C 180,E1 17586.956,E2 17586.956} C_VEL
LIN {X 0,Y 400.257,Z 655.687,A -85,B 0,C 180,E1 17586.33,E2 17586.33} C_VEL
LIN {X 0,Y 398.177,Z 675.511,A -85,B 0,C 180,E1 17585.502,E2 17585.502} C_VEL
LIN {X 0,Y 395.638,Z 695.694,A -85,B 0,C 180,E1 17584.389,E2 17584.389} C_VEL
LIN {X 0,Y 392.895,Z 715.442,A -85,B 0,C 180,E1 17582.996,E2 17582.996} C_VEL
LIN {X 0,Y 390.04,Z 734.256,A -85,B 0,C 180,E1 17581.357,E2 17581.357} C_VEL
LIN {X 0,Y 387.334,Z 751.52,A -85,B 0,C 180,E1 17579.54,E2 17579.54} C_VEL
LIN {X 0,Y 384.645,Z 768.562,A -85,B 0,C 180,E1 17577.393,E2 17577.393} C_VEL
LIN {X 0,Y 382.278,Z 784.065,A -85,B 0,C 180,E1 17575.069,E2 17575.069} C_VEL
LIN {X 0,Y 380.185,Z 798.898,A -85,B 0,C 180,E1 17572.416,E2 17572.416} C_VEL
LIN {X 0,Y 378.593,Z 812.046,A -85,B 0,C 180,E1 17569.597,E2 17569.597} C_VEL
LIN {X 0,Y 377.535,Z 822.936,A -85,B 0,C 180,E1 17566.778,E2 17566.778} C_VEL
LIN {X 0,Y 376.93,Z 831.868,A -85,B 0,C 180,E1 17563.968,E2 17563.968} C_VEL
LIN {X 0,Y 376.66,Z 839.392,A -85,B 0,C 180,E1 17561.018,E2 17561.018} C_VEL
LIN {X 0,Y 376.635,Z 844.855,A -85,B 0,C 180,E1 17558.242,E2 17558.242} C_VEL
LIN {X 0,Y 376.743,Z 848.66,A -85,B 0,C 180,E1 17555.482,E2 17555.482} C_VEL
LIN {X 0,Y 376.858,Z 851.014,A -85,B 0,C 180,E1 17552.585,E2 17552.585} C_VEL
LIN {X 0,Y 376.898,Z 851.734,A -85,B 0,C 180,E1 17549.848,E2 17549.848} C_VEL
LIN {X 0,Y 376.848,Z 850.855,A -85,B 0,C 180,E1 17547.11,E2 17547.11} C_VEL
LIN {X 0,Y 376.723,Z 848.292,A -85,B 0,C 180,E1 17544.212,E2 17544.212} C_VEL
LIN {X 0,Y 376.629,Z 844.329,A -85,B 0,C 180,E1 17541.451,E2 17541.451} C_VEL
LIN {X 0,Y 376.679,Z 838.365,A -85,B 0,C 180,E1 17538.517,E2 17538.517} C_VEL
LIN {X 0,Y 377.01,Z 830.51,A -85,B 0,C 180,E1 17535.565,E2 17535.565} C_VEL
LIN {X 0,Y 377.68,Z 821.222,A -85,B 0,C 180,E1 17532.753,E2 17532.753} C_VEL
LIN {X 0,Y 378.829,Z 809.95,A -85,B 0,C 180,E1 17529.934,E2 17529.934} C_VEL
LIN {X 0,Y 380.405,Z 797.214,A -85,B 0,C 180,E1 17527.271,E2 17527.271} C_VEL
LIN {X 0,Y 382.417,Z 783.045,A -85,B 0,C 180,E1 17524.775,E2 17524.775} C_VEL
LIN {X 0,Y 384.818,Z 767.421,A -85,B 0,C 180,E1 17522.453,E2 17522.453} C_VEL
LIN {X 0,Y 387.539,Z 750.183,A -85,B 0,C 180,E1 17520.307,E2 17520.307} C_VEL
LIN {X 0,Y 390.414,Z 731.886,A -85,B 0,C 180,E1 17518.418,E2 17518.418} C_VEL
LIN {X 0,Y 393.164,Z 713.487,A -85,B 0,C 180,E1 17516.856,E2 17516.856} C_VEL
LIN {X 0,Y 395.788,Z 694.418,A -85,B 0,C 180,E1 17515.538,E2 17515.538} C_VEL
LIN {X 0,Y 398.245,Z 674.689,A -85,B 0,C 180,E1 17514.465,E2 17514.465} C_VEL
LIN {X 0,Y 400.389,Z 653.874,A -85,B 0,C 180,E1 17513.615,E2 17513.615} C_VEL
LIN {X 0,Y 401.888,Z 632.696,A -85,B 0,C 180,E1 17513.008,E2 17513.008} C_VEL
LIN {X 0,Y 409.017,Z 423.458,A -85,B 0,C 180,E1 17508.902,E2 17508.902} C_VEL
LIN {X 0,Y 404.926,Z 380.548,A -85,B 0,C 180,E1 17507.425,E2 17507.425} C_VEL
LIN {X 0,Y 405.115,Z 377.496,A -85,B 0,C 180,E1 17507.14,E2 17507.14} C_VEL
LIN {X 0,Y 398.239,Z 359.716,A -85,B 0,C 180,E1 17504.566,E2 17504.566} C_VEL
LIN {X 0,Y 391.007,Z 343.145,A -85,B 0,C 180,E1 17501.867,E2 17501.867} C_VEL
LIN {X 0,Y 384.173,Z 328.694,A -85,B 0,C 180,E1 17499.23,E2 17499.23} C_VEL
LIN {X 0,Y 379.333,Z 319.376,A -85,B 0,C 180,E1 17497.318,E2 17497.318} C_VEL
LIN {X 0,Y 377.714,Z 315.727,A -85,B 0,C 180,E1 17496.508,E2 17496.508} C_VEL
LIN {X 0,Y 377.672,Z 315.384,A -85,B 0,C 180,E1 17495.064,E2 17495.064} C_VEL
LIN {X 0,Y 377.674,Z 315.425,A -85,B 0,C 180,E1 17491.08,E2 17491.08} C_VEL
LIN {X 0,Y 377.666,Z 315.425,A -85,B 0,C 180,E1 17487.088,E2 17487.088} C_VEL
LIN {X 0,Y 377.66,Z 315.423,A -85,B 0,C 180,E1 17483.068,E2 17483.068} C_VEL
LIN {X 0,Y 377.653,Z 315.424,A -85,B 0,C 180,E1 17479.065,E2 17479.065} C_VEL
LIN {X 0,Y 377.649,Z 315.434,A -85,B 0,C 180,E1 17475.038,E2 17475.038} C_VEL
LIN {X 0,Y 377.645,Z 315.444,A -85,B 0,C 180,E1 17470.989,E2 17470.989} C_VEL
LIN {X 0,Y 377.637,Z 315.43,A -85,B 0,C 180,E1 17466.995,E2 17466.995} C_VEL
LIN {X 0,Y 377.626,Z 315.42,A -85,B 0,C 180,E1 17463.035,E2 17463.035} C_VEL
LIN {X 0,Y 377.621,Z 315.443,A -85,B 0,C 180,E1 17459.089,E2 17459.089} C_VEL
LIN {X 0,Y 377.616,Z 315.441,A -85,B 0,C 180,E1 17455.139,E2 17455.139} C_VEL
LIN {X 0,Y 377.614,Z 315.418,A -85,B 0,C 180,E1 17451.166,E2 17451.166} C_VEL
LIN {X 0,Y 377.621,Z 315.434,A -85,B 0,C 180,E1 17447.149,E2 17447.149} C_VEL
LIN {X 0,Y 377.625,Z 315.445,A -85,B 0,C 180,E1 17443.225,E2 17443.225} C_VEL
LIN {X 0,Y 377.628,Z 315.43,A -85,B 0,C 180,E1 17439.167,E2 17439.167} C_VEL
LIN {X 0,Y 377.631,Z 315.42,A -85,B 0,C 180,E1 17435.103,E2 17435.103} C_VEL
LIN {X 0,Y 377.635,Z 315.429,A -85,B 0,C 180,E1 17431.191,E2 17431.191} C_VEL
LIN {X 0,Y 377.64,Z 315.434,A -85,B 0,C 180,E1 17427.064,E2 17427.064} C_VEL
LIN {X 0,Y 377.643,Z 315.436,A -85,B 0,C 180,E1 17423.057,E2 17423.057} C_VEL
LIN {X 0,Y 377.645,Z 315.431,A -85,B 0,C 180,E1 17418.958,E2 17418.958} C_VEL
LIN {X 0,Y 377.674,Z 315.59,A -85,B 0,C 180,E1 17414.978,E2 17414.978} C_VEL
LIN {X 0,Y 378.967,Z 318.846,A -85,B 0,C 180,E1 17414.14,E2 17414.14} C_VEL
LIN {X 0,Y 383.475,Z 329.131,A -85,B 0,C 180,E1 17411.78,E2 17411.78} C_VEL
LIN {X 0,Y 388.706,Z 341.635,A -85,B 0,C 180,E1 17409.145,E2 17409.145} C_VEL
LIN {X 0,Y 390.668,Z 346.539,A -85,B 0,C 180,E1 17408.243,E2 17408.243} C_VEL
LIN {X 0,Y 401.854,Z 365.241,A -85,B 0,C 180,E1 17406.428,E2 17406.428} C_VEL
LIN {X 0,Y 408.306,Z 377.391,A -85,B 0,C 180,E1 17405.424,E2 17405.424} C_VEL
LIN {X 0,Y 403.778,Z 562.247,A -85,B 0,C 180,E1 17402.19,E2 17402.19} C_VEL
LIN {X 0,Y 402.985,Z 581.209,A -85,B 0,C 180,E1 17401.604,E2 17401.604} C_VEL
LIN {X 0,Y 401.617,Z 599.757,A -85,B 0,C 180,E1 17400.77,E2 17400.77} C_VEL
LIN {X 0,Y 399.777,Z 617.728,A -85,B 0,C 180,E1 17399.682,E2 17399.682} C_VEL
LIN {X 0,Y 397.538,Z 634.563,A -85,B 0,C 180,E1 17398.382,E2 17398.382} C_VEL
LIN {X 0,Y 395.051,Z 650.399,A -85,B 0,C 180,E1 17396.857,E2 17396.857} C_VEL
LIN {X 0,Y 392.371,Z 665.246,A -85,B 0,C 180,E1 17395.105,E2 17395.105} C_VEL
LIN {X 0,Y 389.631,Z 679.059,A -85,B 0,C 180,E1 17393.117,E2 17393.117} C_VEL
LIN {X 0,Y 386.929,Z 691.753,A -85,B 0,C 180,E1 17390.891,E2 17390.891} C_VEL
LIN {X 0,Y 384.473,Z 702.89,A -85,B 0,C 180,E1 17388.498,E2 17388.498} C_VEL
LIN {X 0,Y 382.352,Z 712.53,A -85,B 0,C 180,E1 17385.936,E2 17385.936} C_VEL
LIN {X 0,Y 381.081,Z 718.294,A -85,B 0,C 180,E1 17384.07,E2 17384.07} C_VEL
LIN {X 0,Y 379.485,Z 721.42,A -85,B 0,C 180,E1 17383.02,E2 17383.02} C_VEL
LIN {X 0,Y 372.358,Z 728.649,A -85,B 0,C 180,E1 17380.368,E2 17380.368} C_VEL
LIN {X 0,Y 370.997,Z 730.832,A -85,B 0,C 180,E1 17379.242,E2 17379.242} C_VEL
LIN {X 0,Y 370.207,Z 734.993,A -85,B 0,C 180,E1 17376.202,E2 17376.202} C_VEL
LIN {X 0,Y 369.783,Z 737.5,A -85,B 0,C 180,E1 17373.1,E2 17373.1} C_VEL
LIN {X 0,Y 369.66,Z 738.341,A -85,B 0,C 180,E1 17370,E2 17370} C_VEL
LIN {X 0,Y 369.78,Z 737.558,A -85,B 0,C 180,E1 17366.9,E2 17366.9} C_VEL
LIN {X 0,Y 370.193,Z 735.114,A -85,B 0,C 180,E1 17363.798,E2 17363.798} C_VEL
LIN {X 0,Y 370.996,Z 730.896,A -85,B 0,C 180,E1 17360.694,E2 17360.694} C_VEL
LIN {X 0,Y 372.169,Z 725.135,A -85,B 0,C 180,E1 17357.747,E2 17357.747} C_VEL
LIN {X 0,Y 373.805,Z 717.823,A -85,B 0,C 180,E1 17354.931,E2 17354.931} C_VEL
LIN {X 0,Y 375.895,Z 708.846,A -85,B 0,C 180,E1 17352.226,E2 17352.226} C_VEL
LIN {X 0,Y 378.28,Z 698.604,A -85,B 0,C 180,E1 17349.742,E2 17349.742} C_VEL
LIN {X 0,Y 380.924,Z 687.124,A -85,B 0,C 180,E1 17347.467,E2 17347.467} C_VEL
LIN {X 0,Y 383.827,Z 673.687,A -85,B 0,C 180,E1 17345.286,E2 17345.286} C_VEL
LIN {X 0,Y 386.627,Z 659.727,A -85,B 0,C 180,E1 17343.424,E2 17343.424} C_VEL
LIN {X 0,Y 389.366,Z 644.318,A -85,B 0,C 180,E1 17341.739,E2 17341.739} C_VEL
LIN {X 0,Y 391.951,Z 627.454,A -85,B 0,C 180,E1 17340.254,E2 17340.254} C_VEL
LIN {X 0,Y 394.089,Z 610.146,A -85,B 0,C 180,E1 17339.044,E2 17339.044} C_VEL
LIN {X 0,Y 395.802,Z 591.756,A -85,B 0,C 180,E1 17338.06,E2 17338.06} C_VEL
LIN {X 0,Y 396.944,Z 572.81,A -85,B 0,C 180,E1 17337.329,E2 17337.329} C_VEL
LIN {X 0,Y 397.505,Z 553.125,A -85,B 0,C 180,E1 17336.846,E2 17336.846} C_VEL
LIN {X 0,Y 401.97,Z 379.768,A -85,B 0,C 180,E1 17333.79,E2 17333.79} C_VEL
LIN {X 0,Y 390.796,Z 359.919,A -85,B 0,C 180,E1 17331.972,E2 17331.972} C_VEL
LIN {X 0,Y 382.406,Z 346.181,A -85,B 0,C 180,E1 17330.473,E2 17330.473} C_VEL
LIN {X 0,Y 376.455,Z 331.742,A -85,B 0,C 180,E1 17327.368,E2 17327.368} C_VEL
LIN {X 0,Y 372.549,Z 323.258,A -85,B 0,C 180,E1 17325.334,E2 17325.334} C_VEL
LIN {X 0,Y 370.815,Z 319.53,A -85,B 0,C 180,E1 17324.396,E2 17324.396} C_VEL
LIN {X 0,Y 369.753,Z 316.556,A -85,B 0,C 180,E1 17323.595,E2 17323.595} C_VEL
LIN {X 0,Y 369.738,Z 316.431,A -85,B 0,C 180,E1 17319.585,E2 17319.585} C_VEL
LIN {X 0,Y 369.731,Z 316.428,A -85,B 0,C 180,E1 17315.515,E2 17315.515} C_VEL
LIN {X 0,Y 369.73,Z 316.43,A -85,B 0,C 180,E1 17311.462,E2 17311.462} C_VEL
LIN {X 0,Y 369.73,Z 316.429,A -85,B 0,C 180,E1 17307.504,E2 17307.504} C_VEL
LIN {X 0,Y 369.722,Z 316.417,A -85,B 0,C 180,E1 17303.425,E2 17303.425} C_VEL
LIN {X 0,Y 369.717,Z 316.405,A -85,B 0,C 180,E1 17299.429,E2 17299.429} C_VEL
LIN {X 0,Y 369.715,Z 316.411,A -85,B 0,C 180,E1 17295.369,E2 17295.369} C_VEL
LIN {X 0,Y 369.716,Z 316.432,A -85,B 0,C 180,E1 17291.387,E2 17291.387} C_VEL
LIN {X 0,Y 369.706,Z 316.414,A -85,B 0,C 180,E1 17287.303,E2 17287.303} C_VEL
LIN {X 0,Y 369.699,Z 316.404,A -85,B 0,C 180,E1 17283.256,E2 17283.256} C_VEL
LIN {X 0,Y 369.701,Z 316.426,A -85,B 0,C 180,E1 17279.226,E2 17279.226} C_VEL
LIN {X 0,Y 369.704,Z 316.426,A -85,B 0,C 180,E1 17275.191,E2 17275.191} C_VEL
LIN {X 0,Y 369.707,Z 316.408,A -85,B 0,C 180,E1 17271.133,E2 17271.133} C_VEL
LIN {X 0,Y 369.707,Z 316.407,A -85,B 0,C 180,E1 17267.029,E2 17267.029} C_VEL
LIN {X 0,Y 369.716,Z 316.424,A -85,B 0,C 180,E1 17263.018,E2 17263.018} C_VEL
LIN {X 0,Y 369.718,Z 316.431,A -85,B 0,C 180,E1 17258.905,E2 17258.905} C_VEL
LIN {X 0,Y 369.722,Z 316.433,A -85,B 0,C 180,E1 17254.876,E2 17254.876} C_VEL
LIN {X 0,Y 369.729,Z 316.433,A -85,B 0,C 180,E1 17250.864,E2 17250.864} C_VEL
LIN {X 0,Y 369.733,Z 316.424,A -85,B 0,C 180,E1 17246.889,E2 17246.889} C_VEL
LIN {X 0,Y 369.758,Z 316.563,A -85,B 0,C 180,E1 17244.927,E2 17244.927} C_VEL
LIN {X 0,Y 370.17,Z 318.223,A -85,B 0,C 180,E1 17244.498,E2 17244.498} C_VEL
LIN {X 0,Y 372.351,Z 322.043,A -85,B 0,C 180,E1 17243.599,E2 17243.599} C_VEL
LIN {X 0,Y 378.902,Z 335.083,A -85,B 0,C 180,E1 17240.877,E2 17240.877} C_VEL
LIN {X 0,Y 386.041,Z 350.283,A -85,B 0,C 180,E1 17238.07,E2 17238.07} C_VEL
LIN {X 0,Y 393.187,Z 367.162,A -85,B 0,C 180,E1 17235.322,E2 17235.322} C_VEL
LIN {X 0,Y 398.556,Z 381.111,A -85,B 0,C 180,E1 17233.295,E2 17233.295} C_VEL
LIN {X 0,Y 402.685,Z 425.422,A -85,B 0,C 180,E1 17231.765,E2 17231.765} C_VEL
LIN {X 0,Y 395.21,Z 634.01,A -85,B 0,C 180,E1 17227.611,E2 17227.611} C_VEL
LIN {X 0,Y 393.553,Z 655.231,A -85,B 0,C 180,E1 17226.969,E2 17226.969} C_VEL
LIN {X 0,Y 391.36,Z 675.145,A -85,B 0,C 180,E1 17226.122,E2 17226.122} C_VEL
LIN {X 0,Y 388.72,Z 695.121,A -85,B 0,C 180,E1 17225,E2 17225} C_VEL
LIN {X 0,Y 385.802,Z 715.033,A -85,B 0,C 180,E1 17223.569,E2 17223.569} C_VEL
LIN {X 0,Y 382.721,Z 734.276,A -85,B 0,C 180,E1 17221.851,E2 17221.851} C_VEL
LIN {X 0,Y 379.775,Z 751.99,A -85,B 0,C 180,E1 17219.927,E2 17219.927} C_VEL
LIN {X 0,Y 376.972,Z 768.772,A -85,B 0,C 180,E1 17217.741,E2 17217.741} C_VEL
LIN {X 0,Y 374.578,Z 783.606,A -85,B 0,C 180,E1 17215.451,E2 17215.451} C_VEL
LIN {X 0,Y 372.495,Z 797.539,A -85,B 0,C 180,E1 17212.905,E2 17212.905} C_VEL
LIN {X 0,Y 370.785,Z 810.714,A -85,B 0,C 180,E1 17210.027,E2 17210.027} C_VEL
LIN {X 0,Y 369.64,Z 821.631,A -85,B 0,C 180,E1 17207.147,E2 17207.147} C_VEL
LIN {X 0,Y 368.991,Z 830.591,A -85,B 0,C 180,E1 17204.275,E2 17204.275} C_VEL
LIN {X 0,Y 368.699,Z 838.139,A -85,B 0,C 180,E1 17201.259,E2 17201.259} C_VEL
LIN {X 0,Y 368.68,Z 843.624,A -85,B 0,C 180,E1 17198.421,E2 17198.421} C_VEL
LIN {X 0,Y 368.803,Z 847.442,A -85,B 0,C 180,E1 17195.601,E2 17195.601} C_VEL
LIN {X 0,Y 368.943,Z 849.809,A -85,B 0,C 180,E1 17192.641,E2 17192.641} C_VEL
LIN {X 0,Y 368.989,Z 850.533,A -85,B 0,C 180,E1 17189.845,E2 17189.845} C_VEL
LIN {X 0,Y 368.929,Z 849.649,A -85,B 0,C 180,E1 17187.048,E2 17187.048} C_VEL
LIN {X 0,Y 368.783,Z 847.073,A -85,B 0,C 180,E1 17184.087,E2 17184.087} C_VEL
LIN {X 0,Y 368.677,Z 843.092,A -85,B 0,C 180,E1 17181.265,E2 17181.265} C_VEL
LIN {X 0,Y 368.719,Z 837.108,A -85,B 0,C 180,E1 17178.266,E2 17178.266} C_VEL
LIN {X 0,Y 369.076,Z 829.228,A -85,B 0,C 180,E1 17175.247,E2 17175.247} C_VEL
LIN {X 0,Y 369.794,Z 819.913,A -85,B 0,C 180,E1 17172.373,E2 17172.373} C_VEL
LIN {X 0,Y 371.027,Z 808.611,A -85,B 0,C 180,E1 17169.493,E2 17169.493} C_VEL
LIN {X 0,Y 372.723,Z 795.847,A -85,B 0,C 180,E1 17166.776,E2 17166.776} C_VEL
LIN {X 0,Y 374.873,Z 781.648,A -85,B 0,C 180,E1 17164.231,E2 17164.231} C_VEL
LIN {X 0,Y 377.437,Z 765.979,A -85,B 0,C 180,E1 17161.867,E2 17161.867} C_VEL
LIN {X 0,Y 380.316,Z 748.703,A -85,B 0,C 180,E1 17159.685,E2 17159.685} C_VEL
LIN {X 0,Y 383.337,Z 730.572,A -85,B 0,C 180,E1 17157.79,E2 17157.79} C_VEL
LIN {X 0,Y 386.269,Z 711.874,A -85,B 0,C 180,E1 17156.185,E2 17156.185} C_VEL
LIN {X 0,Y 389.045,Z 692.678,A -85,B 0,C 180,E1 17154.853,E2 17154.853} C_VEL
LIN {X 0,Y 391.54,Z 673.367,A -85,B 0,C 180,E1 17153.799,E2 17153.799} C_VEL
LIN {X 0,Y 393.829,Z 651.904,A -85,B 0,C 180,E1 17152.924,E2 17152.924} C_VEL
LIN {X 0,Y 395.373,Z 629.735,A -85,B 0,C 180,E1 17152.299,E2 17152.299} C_VEL
LIN {X 0,Y 402.659,Z 424.289,A -85,B 0,C 180,E1 17148.22,E2 17148.22} C_VEL
LIN {X 0,Y 398.425,Z 380.897,A -85,B 0,C 180,E1 17146.699,E2 17146.699} C_VEL
LIN {X 0,Y 391.232,Z 362.281,A -85,B 0,C 180,E1 17143.936,E2 17143.936} C_VEL
LIN {X 0,Y 383.727,Z 345.139,A -85,B 0,C 180,E1 17141.043,E2 17141.043} C_VEL
LIN {X 0,Y 377.601,Z 332.574,A -85,B 0,C 180,E1 17138.637,E2 17138.637} C_VEL
LIN {X 0,Y 373.7,Z 324.765,A -85,B 0,C 180,E1 17137.013,E2 17137.013} C_VEL
LIN {X 0,Y 371.587,Z 320.616,A -85,B 0,C 180,E1 17136.106,E2 17136.106} C_VEL
LIN {X 0,Y 369.853,Z 317.138,A -85,B 0,C 180,E1 17135.32,E2 17135.32} C_VEL
LIN {X 0,Y 369.741,Z 316.427,A -85,B 0,C 180,E1 17134.98,E2 17134.98} C_VEL
LIN {X 0,Y 369.745,Z 316.412,A -85,B 0,C 180,E1 17130.917,E2 17130.917} C_VEL
LIN {X 0,Y 369.741,Z 316.412,A -85,B 0,C 180,E1 17126.828,E2 17126.828} C_VEL
LIN {X 0,Y 369.745,Z 316.408,A -85,B 0,C 180,E1 17122.749,E2 17122.749} C_VEL
LIN {X 0,Y 369.732,Z 316.407,A -85,B 0,C 180,E1 17118.608,E2 17118.608} C_VEL
LIN {X 0,Y 369.73,Z 316.41,A -85,B 0,C 180,E1 17114.509,E2 17114.509} C_VEL
LIN {X 0,Y 369.719,Z 316.429,A -85,B 0,C 180,E1 17110.439,E2 17110.439} C_VEL
LIN {X 0,Y 369.718,Z 316.424,A -85,B 0,C 180,E1 17106.366,E2 17106.366} C_VEL
LIN {X 0,Y 369.707,Z 316.406,A -85,B 0,C 180,E1 17102.325,E2 17102.325} C_VEL
LIN {X 0,Y 369.704,Z 316.414,A -85,B 0,C 180,E1 17098.295,E2 17098.295} C_VEL
LIN {X 0,Y 369.7,Z 316.434,A -85,B 0,C 180,E1 17094.101,E2 17094.101} C_VEL
LIN {X 0,Y 369.709,Z 316.411,A -85,B 0,C 180,E1 17090.19,E2 17090.19} C_VEL
LIN {X 0,Y 369.708,Z 316.404,A -85,B 0,C 180,E1 17086.072,E2 17086.072} C_VEL
LIN {X 0,Y 369.717,Z 316.423,A -85,B 0,C 180,E1 17082.043,E2 17082.043} C_VEL
LIN {X 0,Y 369.717,Z 316.433,A -85,B 0,C 180,E1 17077.919,E2 17077.919} C_VEL
LIN {X 0,Y 369.718,Z 316.419,A -85,B 0,C 180,E1 17073.844,E2 17073.844} C_VEL
LIN {X 0,Y 369.731,Z 316.411,A -85,B 0,C 180,E1 17069.922,E2 17069.922} C_VEL
LIN {X 0,Y 369.73,Z 316.412,A -85,B 0,C 180,E1 17065.842,E2 17065.842} C_VEL
LIN {X 0,Y 369.73,Z 316.415,A -85,B 0,C 180,E1 17061.736,E2 17061.736} C_VEL
LIN {X 0,Y 369.732,Z 316.419,A -85,B 0,C 180,E1 17057.672,E2 17057.672} C_VEL
LIN {X 0,Y 369.783,Z 316.727,A -85,B 0,C 180,E1 17056.195,E2 17056.195} C_VEL
LIN {X 0,Y 371.162,Z 320.086,A -85,B 0,C 180,E1 17055.323,E2 17055.323} C_VEL
LIN {X 0,Y 375.606,Z 329.93,A -85,B 0,C 180,E1 17052.941,E2 17052.941} C_VEL
LIN {X 0,Y 381.065,Z 342.824,A -85,B 0,C 180,E1 17050.105,E2 17050.105} C_VEL
LIN {X 0,Y 382.832,Z 347.151,A -85,B 0,C 180,E1 17049.28,E2 17049.28} C_VEL
LIN {X 0,Y 394.094,Z 365.545,A -85,B 0,C 180,E1 17047.368,E2 17047.368} C_VEL
LIN {X 0,Y 402.008,Z 380.162,A -85,B 0,C 180,E1 17046.09,E2 17046.09} C_VEL
LIN {X 0,Y 397.256,Z 562.922,A -85,B 0,C 180,E1 17042.846,E2 17042.846} C_VEL
LIN {X 0,Y 396.432,Z 581.766,A -85,B 0,C 180,E1 17042.258,E2 17042.258} C_VEL
LIN {X 0,Y 395.024,Z 600.147,A -85,B 0,C 180,E1 17041.426,E2 17041.426} C_VEL
LIN {X 0,Y 393.223,Z 617.149,A -85,B 0,C 180,E1 17040.397,E2 17040.397} C_VEL
LIN {X 0,Y 391.012,Z 633.44,A -85,B 0,C 180,E1 17039.151,E2 17039.151} C_VEL
LIN {X 0,Y 388.517,Z 648.98,A -85,B 0,C 180,E1 17037.678,E2 17037.678} C_VEL
LIN {X 0,Y 385.67,Z 664.336,A -85,B 0,C 180,E1 17035.893,E2 17035.893} C_VEL
LIN {X 0,Y 382.777,Z 678.445,A -85,B 0,C 180,E1 17033.883,E2 17033.883} C_VEL
LIN {X 0,Y 380.077,Z 690.644,A -85,B 0,C 180,E1 17031.772,E2 17031.772} C_VEL
LIN {X 0,Y 377.41,Z 702.183,A -85,B 0,C 180,E1 17029.338,E2 17029.338} C_VEL
LIN {X 0,Y 375.092,Z 712.176,A -85,B 0,C 180,E1 17026.731,E2 17026.731} C_VEL
LIN {X 0,Y 373.137,Z 720.642,A -85,B 0,C 180,E1 17023.955,E2 17023.955} C_VEL
LIN {X 0,Y 371.641,Z 727.555,A -85,B 0,C 180,E1 17021.012,E2 17021.012} C_VEL
LIN {X 0,Y 370.997,Z 730.832,A -85,B 0,C 180,E1 17019.242,E2 17019.242} C_VEL
LIN {X 0,Y 369.69,Z 732.861,A -85,B 0,C 180,E1 17018.1,E2 17018.1} C_VEL
LIN {X 0,Y 364.253,Z 736.462,A -85,B 0,C 180,E1 17015.777,E2 17015.777} C_VEL
LIN {X 0,Y 362.158,Z 737.879,A -85,B 0,C 180,E1 17014.424,E2 17014.424} C_VEL
LIN {X 0,Y 361.958,Z 738.178,A -85,B 0,C 180,E1 17013.987,E2 17013.987} C_VEL
LIN {X 0,Y 361.753,Z 739.441,A -85,B 0,C 180,E1 17010.792,E2 17010.792} C_VEL
LIN {X 0,Y 361.816,Z 739.062,A -85,B 0,C 180,E1 17007.624,E2 17007.624} C_VEL
LIN {X 0,Y 362.17,Z 737.043,A -85,B 0,C 180,E1 17004.455,E2 17004.455} C_VEL
LIN {X 0,Y 362.911,Z 733.295,A -85,B 0,C 180,E1 17001.285,E2 17001.285} C_VEL
LIN {X 0,Y 364.039,Z 728.011,A -85,B 0,C 180,E1 16998.274,E2 16998.274} C_VEL
LIN {X 0,Y 365.698,Z 720.873,A -85,B 0,C 180,E1 16995.27,E2 16995.27} C_VEL
LIN {X 0,Y 367.704,Z 712.688,A -85,B 0,C 180,E1 16992.596,E2 16992.596} C_VEL
LIN {X 0,Y 370.188,Z 702.54,A -85,B 0,C 180,E1 16989.94,E2 16989.94} C_VEL
LIN {X 0,Y 373.036,Z 690.826,A -85,B 0,C 180,E1 16987.463,E2 16987.463} C_VEL
LIN {X 0,Y 375.895,Z 678.427,A -85,B 0,C 180,E1 16985.317,E2 16985.317} C_VEL
LIN {X 0,Y 378.848,Z 664.599,A -85,B 0,C 180,E1 16983.343,E2 16983.343} C_VEL
LIN {X 0,Y 381.823,Z 649.137,A -85,B 0,C 180,E1 16981.538,E2 16981.538} C_VEL
LIN {X 0,Y 384.454,Z 633.384,A -85,B 0,C 180,E1 16980.045,E2 16980.045} C_VEL
LIN {X 0,Y 386.892,Z 615.704,A -85,B 0,C 180,E1 16978.706,E2 16978.706} C_VEL
LIN {X 0,Y 388.777,Z 597.903,A -85,B 0,C 180,E1 16977.662,E2 16977.662} C_VEL
LIN {X 0,Y 390.173,Z 578.929,A -85,B 0,C 180,E1 16976.843,E2 16976.843} C_VEL
LIN {X 0,Y 390.918,Z 559.61,A -85,B 0,C 180,E1 16976.286,E2 16976.286} C_VEL
LIN {X 0,Y 395.719,Z 382.656,A -85,B 0,C 180,E1 16973.102,E2 16973.102} C_VEL
LIN {X 0,Y 385.088,Z 363.871,A -85,B 0,C 180,E1 16971.312,E2 16971.312} C_VEL
LIN {X 0,Y 374.883,Z 347.475,A -85,B 0,C 180,E1 16969.476,E2 16969.476} C_VEL
LIN {X 0,Y 368.778,Z 333.08,A -85,B 0,C 180,E1 16966.263,E2 16966.263} C_VEL
LIN {X 0,Y 364.779,Z 324.491,A -85,B 0,C 180,E1 16964.101,E2 16964.101} C_VEL
LIN {X 0,Y 363.332,Z 321.242,A -85,B 0,C 180,E1 16963.254,E2 16963.254} C_VEL
LIN {X 0,Y 361.83,Z 317.634,A -85,B 0,C 180,E1 16962.249,E2 16962.249} C_VEL
LIN {X 0,Y 361.794,Z 317.402,A -85,B 0,C 180,E1 16958.247,E2 16958.247} C_VEL
LIN {X 0,Y 361.794,Z 317.399,A -85,B 0,C 180,E1 16954.126,E2 16954.126} C_VEL
LIN {X 0,Y 361.798,Z 317.397,A -85,B 0,C 180,E1 16950.014,E2 16950.014} C_VEL
LIN {X 0,Y 361.795,Z 317.401,A -85,B 0,C 180,E1 16945.891,E2 16945.891} C_VEL
LIN {X 0,Y 361.807,Z 317.415,A -85,B 0,C 180,E1 16941.735,E2 16941.735} C_VEL
LIN {X 0,Y 361.789,Z 317.414,A -85,B 0,C 180,E1 16937.532,E2 16937.532} C_VEL
LIN {X 0,Y 361.777,Z 317.395,A -85,B 0,C 180,E1 16933.392,E2 16933.392} C_VEL
LIN {X 0,Y 361.771,Z 317.393,A -85,B 0,C 180,E1 16929.375,E2 16929.375} C_VEL
LIN {X 0,Y 361.774,Z 317.42,A -85,B 0,C 180,E1 16925.392,E2 16925.392} C_VEL
LIN {X 0,Y 361.762,Z 317.407,A -85,B 0,C 180,E1 16921.267,E2 16921.267} C_VEL
LIN {X 0,Y 361.757,Z 317.392,A -85,B 0,C 180,E1 16917.149,E2 16917.149} C_VEL
LIN {X 0,Y 361.758,Z 317.404,A -85,B 0,C 180,E1 16913.015,E2 16913.015} C_VEL
LIN {X 0,Y 361.766,Z 317.422,A -85,B 0,C 180,E1 16909.006,E2 16909.006} C_VEL
LIN {X 0,Y 361.767,Z 317.41,A -85,B 0,C 180,E1 16904.942,E2 16904.942} C_VEL
LIN {X 0,Y 361.773,Z 317.4,A -85,B 0,C 180,E1 16900.941,E2 16900.941} C_VEL
LIN {X 0,Y 361.779,Z 317.398,A -85,B 0,C 180,E1 16896.893,E2 16896.893} C_VEL
LIN {X 0,Y 361.784,Z 317.4,A -85,B 0,C 180,E1 16892.858,E2 16892.858} C_VEL
LIN {X 0,Y 361.793,Z 317.401,A -85,B 0,C 180,E1 16888.883,E2 16888.883} C_VEL
LIN {X 0,Y 361.809,Z 317.689,A -85,B 0,C 180,E1 16886.283,E2 16886.283} C_VEL
LIN {X 0,Y 363.225,Z 321.045,A -85,B 0,C 180,E1 16885.455,E2 16885.455} C_VEL
LIN {X 0,Y 364.353,Z 322.737,A -85,B 0,C 180,E1 16885.003,E2 16885.003} C_VEL
LIN {X 0,Y 366.44,Z 326.654,A -85,B 0,C 180,E1 16884.081,E2 16884.081} C_VEL
LIN {X 0,Y 373.538,Z 341.123,A -85,B 0,C 180,E1 16881.022,E2 16881.022} C_VEL
LIN {X 0,Y 380.254,Z 355.639,A -85,B 0,C 180,E1 16878.299,E2 16878.299} C_VEL
LIN {X 0,Y 387.27,Z 372.531,A -85,B 0,C 180,E1 16875.496,E2 16875.496} C_VEL
LIN {X 0,Y 390.404,Z 380.571,A -85,B 0,C 180,E1 16874.316,E2 16874.316} C_VEL
LIN {X 0,Y 392.72,Z 385.25,A -85,B 0,C 180,E1 16873.91,E2 16873.91} C_VEL
LIN {X 0,Y 396.383,Z 426.827,A -85,B 0,C 180,E1 16872.457,E2 16872.457} C_VEL
LIN {X 0,Y 388.623,Z 633.809,A -85,B 0,C 180,E1 16868.28,E2 16868.28} C_VEL
LIN {X 0,Y 386.828,Z 655.575,A -85,B 0,C 180,E1 16867.604,E2 16867.604} C_VEL
LIN {X 0,Y 384.509,Z 675.463,A -85,B 0,C 180,E1 16866.731,E2 16866.731} C_VEL
LIN {X 0,Y 381.867,Z 694.456,A -85,B 0,C 180,E1 16865.639,E2 16865.639} C_VEL
LIN {X 0,Y 378.833,Z 714.109,A -85,B 0,C 180,E1 16864.205,E2 16864.205} C_VEL
LIN {X 0,Y 375.571,Z 733.516,A -85,B 0,C 180,E1 16862.443,E2 16862.443} C_VEL
LIN {X 0,Y 372.347,Z 751.824,A -85,B 0,C 180,E1 16860.408,E2 16860.408} C_VEL
LIN {X 0,Y 369.411,Z 768.447,A -85,B 0,C 180,E1 16858.183,E2 16858.183} C_VEL
LIN {X 0,Y 366.894,Z 783.145,A -85,B 0,C 180,E1 16855.85,E2 16855.85} C_VEL
LIN {X 0,Y 364.705,Z 796.986,A -85,B 0,C 180,E1 16853.252,E2 16853.252} C_VEL
LIN {X 0,Y 362.907,Z 810.07,A -85,B 0,C 180,E1 16850.312,E2 16850.312} C_VEL
LIN {X 0,Y 361.65,Z 821.465,A -85,B 0,C 180,E1 16847.206,E2 16847.206} C_VEL
LIN {X 0,Y 360.973,Z 830.671,A -85,B 0,C 180,E1 16844.108,E2 16844.108} C_VEL
LIN {X 0,Y 360.722,Z 837.916,A -85,B 0,C 180,E1 16841.026,E2 16841.026} C_VEL
LIN {X 0,Y 360.753,Z 843.342,A -85,B 0,C 180,E1 16837.965,E2 16837.965} C_VEL
LIN {X 0,Y 360.901,Z 846.9,A -85,B 0,C 180,E1 16835.086,E2 16835.086} C_VEL
LIN {X 0,Y 361.035,Z 848.838,A -85,B 0,C 180,E1 16832.222,E2 16832.222} C_VEL
LIN {X 0,Y 361.073,Z 849.256,A -85,B 0,C 180,E1 16829.365,E2 16829.365} C_VEL
LIN {X 0,Y 360.979,Z 848.194,A -85,B 0,C 180,E1 16826.506,E2 16826.506} C_VEL
LIN {X 0,Y 360.83,Z 845.488,A -85,B 0,C 180,E1 16823.636,E2 16823.636} C_VEL
LIN {X 0,Y 360.721,Z 840.992,A -85,B 0,C 180,E1 16820.588,E2 16820.588} C_VEL
LIN {X 0,Y 360.775,Z 835.116,A -85,B 0,C 180,E1 16817.679,E2 16817.679} C_VEL
LIN {X 0,Y 361.203,Z 827.04,A -85,B 0,C 180,E1 16814.589,E2 16814.589} C_VEL
LIN {X 0,Y 362.032,Z 817.468,A -85,B 0,C 180,E1 16811.649,E2 16811.649} C_VEL
LIN {X 0,Y 363.331,Z 806.583,A -85,B 0,C 180,E1 16808.87,E2 16808.87} C_VEL
LIN {X 0,Y 365.194,Z 793.65,A -85,B 0,C 180,E1 16806.097,E2 16806.097} C_VEL
LIN {X 0,Y 367.529,Z 779.26,A -85,B 0,C 180,E1 16803.503,E2 16803.503} C_VEL
LIN {X 0,Y 370.249,Z 763.693,A -85,B 0,C 180,E1 16801.143,E2 16801.143} C_VEL
LIN {X 0,Y 373.268,Z 746.52,A -85,B 0,C 180,E1 16798.961,E2 16798.961} C_VEL
LIN {X 0,Y 376.417,Z 728.601,A -85,B 0,C 180,E1 16797.074,E2 16797.074} C_VEL
LIN {X 0,Y 379.598,Z 709.338,A -85,B 0,C 180,E1 16795.416,E2 16795.416} C_VEL
LIN {X 0,Y 382.536,Z 689.796,A -85,B 0,C 180,E1 16794.072,E2 16794.072} C_VEL
LIN {X 0,Y 385.131,Z 670.054,A -85,B 0,C 180,E1 16793.012,E2 16793.012} C_VEL
LIN {X 0,Y 387.372,Z 649.543,A -85,B 0,C 180,E1 16792.197,E2 16792.197} C_VEL
LIN {X 0,Y 388.855,Z 628.164,A -85,B 0,C 180,E1 16791.598,E2 16791.598} C_VEL
LIN {X 0,Y 396.355,Z 425.215,A -85,B 0,C 180,E1 16787.517,E2 16787.517} C_VEL
LIN {X 0,Y 392.46,Z 384.426,A -85,B 0,C 180,E1 16786.057,E2 16786.057} C_VEL
LIN {X 0,Y 389.67,Z 378.987,A -85,B 0,C 180,E1 16785.506,E2 16785.506} C_VEL
LIN {X 0,Y 383.271,Z 362.639,A -85,B 0,C 180,E1 16782.912,E2 16782.912} C_VEL
LIN {X 0,Y 376.067,Z 346.399,A -85,B 0,C 180,E1 16780.032,E2 16780.032} C_VEL
LIN {X 0,Y 370.219,Z 334.377,A -85,B 0,C 180,E1 16777.615,E2 16777.615} C_VEL
LIN {X 0,Y 365.908,Z 325.96,A -85,B 0,C 180,E1 16775.753,E2 16775.753} C_VEL
LIN {X 0,Y 363.974,Z 321.946,A -85,B 0,C 180,E1 16774.847,E2 16774.847} C_VEL
LIN {X 0,Y 362.14,Z 318.988,A -85,B 0,C 180,E1 16774.079,E2 16774.079} C_VEL
LIN {X 0,Y 361.774,Z 317.425,A -85,B 0,C 180,E1 16773.623,E2 16773.623} C_VEL
LIN {X 0,Y 361.774,Z 317.422,A -85,B 0,C 180,E1 16769.468,E2 16769.468} C_VEL
LIN {X 0,Y 361.772,Z 317.424,A -85,B 0,C 180,E1 16765.347,E2 16765.347} C_VEL
LIN {X 0,Y 361.767,Z 317.419,A -85,B 0,C 180,E1 16761.349,E2 16761.349} C_VEL
LIN {X 0,Y 361.756,Z 317.407,A -85,B 0,C 180,E1 16757.367,E2 16757.367} C_VEL
LIN {X 0,Y 361.75,Z 317.396,A -85,B 0,C 180,E1 16753.374,E2 16753.374} C_VEL
LIN {X 0,Y 361.747,Z 317.404,A -85,B 0,C 180,E1 16749.352,E2 16749.352} C_VEL
LIN {X 0,Y 361.743,Z 317.425,A -85,B 0,C 180,E1 16745.392,E2 16745.392} C_VEL
LIN {X 0,Y 361.738,Z 317.411,A -85,B 0,C 180,E1 16741.267,E2 16741.267} C_VEL
LIN {X 0,Y 361.734,Z 317.395,A -85,B 0,C 180,E1 16737.148,E2 16737.148} C_VEL
LIN {X 0,Y 361.738,Z 317.416,A -85,B 0,C 180,E1 16733.174,E2 16733.174} C_VEL
LIN {X 0,Y 361.749,Z 317.422,A -85,B 0,C 180,E1 16729.005,E2 16729.005} C_VEL
LIN {X 0,Y 361.751,Z 317.398,A -85,B 0,C 180,E1 16724.941,E2 16724.941} C_VEL
LIN {X 0,Y 361.755,Z 317.398,A -85,B 0,C 180,E1 16720.949,E2 16720.949} C_VEL
LIN {X 0,Y 361.76,Z 317.414,A -85,B 0,C 180,E1 16716.891,E2 16716.891} C_VEL
LIN {X 0,Y 361.765,Z 317.423,A -85,B 0,C 180,E1 16712.864,E2 16712.864} C_VEL
LIN {X 0,Y 361.764,Z 317.417,A -85,B 0,C 180,E1 16708.879,E2 16708.879} C_VEL
LIN {X 0,Y 361.772,Z 317.415,A -85,B 0,C 180,E1 16704.716,E2 16704.716} C_VEL
LIN {X 0,Y 361.776,Z 317.417,A -85,B 0,C 180,E1 16700.699,E2 16700.699} C_VEL
LIN {X 0,Y 361.828,Z 317.682,A -85,B 0,C 180,E1 16697.603,E2 16697.603} C_VEL
LIN {X 0,Y 363.111,Z 320.945,A -85,B 0,C 180,E1 16696.713,E2 16696.713} C_VEL
LIN {X 0,Y 364.066,Z 322.79,A -85,B 0,C 180,E1 16696.204,E2 16696.204} C_VEL
LIN {X 0,Y 369.244,Z 334.106,A -85,B 0,C 180,E1 16693.359,E2 16693.359} C_VEL
LIN {X 0,Y 374.977,Z 347.675,A -85,B 0,C 180,E1 16690.386,E2 16690.386} C_VEL
LIN {X 0,Y 387.256,Z 367.582,A -85,B 0,C 180,E1 16688.198,E2 16688.198} C_VEL
LIN {X 0,Y 395.768,Z 382.959,A -85,B 0,C 180,E1 16686.776,E2 16686.776} C_VEL
LIN {X 0,Y 390.787,Z 563.632,A -85,B 0,C 180,E1 16683.522,E2 16683.522} C_VEL
LIN {X 0,Y 389.925,Z 582.444,A -85,B 0,C 180,E1 16682.929,E2 16682.929} C_VEL
LIN {X 0,Y 388.497,Z 600.381,A -85,B 0,C 180,E1 16682.112,E2 16682.112} C_VEL
LIN {X 0,Y 386.602,Z 617.669,A -85,B 0,C 180,E1 16681.061,E2 16681.061} C_VEL
LIN {X 0,Y 384.298,Z 634.059,A -85,B 0,C 180,E1 16679.797,E2 16679.797} C_VEL
LIN {X 0,Y 381.56,Z 650.388,A -85,B 0,C 180,E1 16678.228,E2 16678.228} C_VEL
LIN {X 0,Y 378.602,Z 665.622,A -85,B 0,C 180,E1 16676.422,E2 16676.422} C_VEL
LIN {X 0,Y 375.567,Z 679.75,A -85,B 0,C 180,E1 16674.371,E2 16674.371} C_VEL
LIN {X 0,Y 372.742,Z 691.919,A -85,B 0,C 180,E1 16672.223,E2 16672.223} C_VEL
LIN {X 0,Y 369.945,Z 703.438,A -85,B 0,C 180,E1 16669.745,E2 16669.745} C_VEL
LIN {X 0,Y 367.507,Z 713.414,A -85,B 0,C 180,E1 16667.087,E2 16667.087} C_VEL
LIN {X 0,Y 365.445,Z 721.869,A -85,B 0,C 180,E1 16664.255,E2 16664.255} C_VEL
LIN {X 0,Y 363.93,Z 728.45,A -85,B 0,C 180,E1 16661.409,E2 16661.409} C_VEL
LIN {X 0,Y 362.838,Z 733.614,A -85,B 0,C 180,E1 16658.393,E2 16658.393} C_VEL
LIN {X 0,Y 362.132,Z 737.234,A -85,B 0,C 180,E1 16655.228,E2 16655.228} C_VEL
LIN {X 0,Y 361.958,Z 738.178,A -85,B 0,C 180,E1 16653.987,E2 16653.987} C_VEL
LIN {X 0,Y 360.846,Z 739.026,A -85,B 0,C 180,E1 16652.776,E2 16652.776} C_VEL
LIN {X 0,Y 354.676,Z 740.6,A -85,B 0,C 180,E1 16649.615,E2 16649.615} C_VEL
LIN {X 0,Y 353.866,Z 740.566,A -85,B 0,C 180,E1 16648.451,E2 16648.451} C_VEL
LIN {X 0,Y 354.168,Z 738.956,A -85,B 0,C 180,E1 16645.142,E2 16645.142} C_VEL
LIN {X 0,Y 354.843,Z 735.653,A -85,B 0,C 180,E1 16641.901,E2 16641.901} C_VEL
LIN {X 0,Y 355.983,Z 730.512,A -85,B 0,C 180,E1 16638.662,E2 16638.662} C_VEL
LIN {X 0,Y 357.614,Z 723.781,A -85,B 0,C 180,E1 16635.592,E2 16635.592} C_VEL
LIN {X 0,Y 359.742,Z 715.516,A -85,B 0,C 180,E1 16632.699,E2 16632.699} C_VEL
LIN {X 0,Y 362.259,Z 705.753,A -85,B 0,C 180,E1 16629.987,E2 16629.987} C_VEL
LIN {X 0,Y 365.146,Z 694.482,A -85,B 0,C 180,E1 16627.459,E2 16627.459} C_VEL
LIN {X 0,Y 368.067,Z 682.609,A -85,B 0,C 180,E1 16625.271,E2 16625.271} C_VEL
LIN {X 0,Y 371.207,Z 668.841,A -85,B 0,C 180,E1 16623.182,E2 16623.182} C_VEL
LIN {X 0,Y 374.271,Z 654.067,A -85,B 0,C 180,E1 16621.346,E2 16621.346} C_VEL
LIN {X 0,Y 377.109,Z 638.352,A -85,B 0,C 180,E1 16619.752,E2 16619.752} C_VEL
LIN {X 0,Y 379.653,Z 621.703,A -85,B 0,C 180,E1 16618.394,E2 16618.394} C_VEL
LIN {X 0,Y 381.841,Z 603.378,A -85,B 0,C 180,E1 16617.224,E2 16617.224} C_VEL
LIN {X 0,Y 383.453,Z 584.426,A -85,B 0,C 180,E1 16616.325,E2 16616.325} C_VEL
LIN {X 0,Y 384.412,Z 565.234,A -85,B 0,C 180,E1 16615.699,E2 16615.699} C_VEL
LIN {X 0,Y 386.262,Z 495.829,A -85,B 0,C 180,E1 16614.403,E2 16614.403} C_VEL
LIN {X 0,Y 389.523,Z 385.592,A -85,B 0,C 180,E1 16612.393,E2 16612.393} C_VEL
LIN {X 0,Y 378.787,Z 366.622,A -85,B 0,C 180,E1 16610.513,E2 16610.513} C_VEL
LIN {X 0,Y 367.094,Z 348.215,A -85,B 0,C 180,E1 16608.32,E2 16608.32} C_VEL
LIN {X 0,Y 361.38,Z 334.825,A -85,B 0,C 180,E1 16605.209,E2 16605.209} C_VEL
LIN {X 0,Y 357.156,Z 326.047,A -85,B 0,C 180,E1 16602.866,E2 16602.866} C_VEL
LIN {X 0,Y 355.397,Z 322.186,A -85,B 0,C 180,E1 16601.797,E2 16601.797} C_VEL
LIN {X 0,Y 353.872,Z 318.649,A -85,B 0,C 180,E1 16600.745,E2 16600.745} C_VEL
LIN {X 0,Y 353.833,Z 318.398,A -85,B 0,C 180,E1 16596.804,E2 16596.804} C_VEL
LIN {X 0,Y 353.83,Z 318.399,A -85,B 0,C 180,E1 16592.641,E2 16592.641} C_VEL
LIN {X 0,Y 353.83,Z 318.393,A -85,B 0,C 180,E1 16588.502,E2 16588.502} C_VEL
LIN {X 0,Y 353.828,Z 318.384,A -85,B 0,C 180,E1 16584.367,E2 16584.367} C_VEL
LIN {X 0,Y 353.826,Z 318.385,A -85,B 0,C 180,E1 16580.256,E2 16580.256} C_VEL
LIN {X 0,Y 353.831,Z 318.4,A -85,B 0,C 180,E1 16576.077,E2 16576.077} C_VEL
LIN {X 0,Y 353.833,Z 318.407,A -85,B 0,C 180,E1 16571.905,E2 16571.905} C_VEL
LIN {X 0,Y 353.848,Z 318.382,A -85,B 0,C 180,E1 16567.632,E2 16567.632} C_VEL
LIN {X 0,Y 353.827,Z 318.38,A -85,B 0,C 180,E1 16563.402,E2 16563.402} C_VEL
LIN {X 0,Y 353.82,Z 318.403,A -85,B 0,C 180,E1 16559.191,E2 16559.191} C_VEL
LIN {X 0,Y 353.813,Z 318.409,A -85,B 0,C 180,E1 16554.975,E2 16554.975} C_VEL
LIN {X 0,Y 353.815,Z 318.387,A -85,B 0,C 180,E1 16550.895,E2 16550.895} C_VEL
LIN {X 0,Y 353.815,Z 318.384,A -85,B 0,C 180,E1 16546.768,E2 16546.768} C_VEL
LIN {X 0,Y 353.821,Z 318.397,A -85,B 0,C 180,E1 16542.74,E2 16542.74} C_VEL
LIN {X 0,Y 353.824,Z 318.407,A -85,B 0,C 180,E1 16538.621,E2 16538.621} C_VEL
LIN {X 0,Y 353.829,Z 318.411,A -85,B 0,C 180,E1 16534.563,E2 16534.563} C_VEL
LIN {X 0,Y 353.827,Z 318.405,A -85,B 0,C 180,E1 16530.362,E2 16530.362} C_VEL
LIN {X 0,Y 353.867,Z 318.641,A -85,B 0,C 180,E1 16527.844,E2 16527.844} C_VEL
LIN {X 0,Y 355.335,Z 322.13,A -85,B 0,C 180,E1 16526.915,E2 16526.915} C_VEL
LIN {X 0,Y 356.543,Z 324.006,A -85,B 0,C 180,E1 16526.393,E2 16526.393} C_VEL
LIN {X 0,Y 359.087,Z 328.882,A -85,B 0,C 180,E1 16525.194,E2 16525.194} C_VEL
LIN {X 0,Y 363.891,Z 338.413,A -85,B 0,C 180,E1 16523.006,E2 16523.006} C_VEL
LIN {X 0,Y 370.158,Z 351.303,A -85,B 0,C 180,E1 16520.337,E2 16520.337} C_VEL
LIN {X 0,Y 377.444,Z 368.019,A -85,B 0,C 180,E1 16517.301,E2 16517.301} C_VEL
LIN {X 0,Y 382.211,Z 379.875,A -85,B 0,C 180,E1 16515.407,E2 16515.407} C_VEL
LIN {X 0,Y 386.858,Z 388.891,A -85,B 0,C 180,E1 16514.566,E2 16514.566} C_VEL
LIN {X 0,Y 390.151,Z 428.02,A -85,B 0,C 180,E1 16513.175,E2 16513.175} C_VEL
LIN {X 0,Y 382.1,Z 633.428,A -85,B 0,C 180,E1 16508.976,E2 16508.976} C_VEL
LIN {X 0,Y 380.185,Z 655.538,A -85,B 0,C 180,E1 16508.273,E2 16508.273} C_VEL
LIN {X 0,Y 377.611,Z 676.539,A -85,B 0,C 180,E1 16507.325,E2 16507.325} C_VEL
LIN {X 0,Y 374.68,Z 696.317,A -85,B 0,C 180,E1 16506.138,E2 16506.138} C_VEL
LIN {X 0,Y 371.564,Z 715.319,A -85,B 0,C 180,E1 16504.689,E2 16504.689} C_VEL
LIN {X 0,Y 368.342,Z 733.432,A -85,B 0,C 180,E1 16502.99,E2 16502.99} C_VEL
LIN {X 0,Y 365.059,Z 751.037,A -85,B 0,C 180,E1 16500.989,E2 16500.989} C_VEL
LIN {X 0,Y 361.872,Z 768.129,A -85,B 0,C 180,E1 16498.644,E2 16498.644} C_VEL
LIN {X 0,Y 359.067,Z 783.6,A -85,B 0,C 180,E1 16496.101,E2 16496.101} C_VEL
LIN {X 0,Y 356.801,Z 797.175,A -85,B 0,C 180,E1 16493.448,E2 16493.448} C_VEL
LIN {X 0,Y 355.032,Z 809.393,A -85,B 0,C 180,E1 16490.611,E2 16490.611} C_VEL
LIN {X 0,Y 353.768,Z 820.169,A -85,B 0,C 180,E1 16487.602,E2 16487.602} C_VEL
LIN {X 0,Y 353.035,Z 829.399,A -85,B 0,C 180,E1 16484.432,E2 16484.432} C_VEL
LIN {X 0,Y 352.76,Z 836.669,A -85,B 0,C 180,E1 16481.277,E2 16481.277} C_VEL
LIN {X 0,Y 352.798,Z 842.114,A -85,B 0,C 180,E1 16478.146,E2 16478.146} C_VEL
LIN {X 0,Y 352.969,Z 845.688,A -85,B 0,C 180,E1 16475.201,E2 16475.201} C_VEL
LIN {X 0,Y 353.121,Z 847.634,A -85,B 0,C 180,E1 16472.272,E2 16472.272} C_VEL
LIN {X 0,Y 353.163,Z 848.054,A -85,B 0,C 180,E1 16469.351,E2 16469.351} C_VEL
LIN {X 0,Y 353.058,Z 846.987,A -85,B 0,C 180,E1 16466.428,E2 16466.428} C_VEL
LIN {X 0,Y 352.892,Z 844.269,A -85,B 0,C 180,E1 16463.493,E2 16463.493} C_VEL
LIN {X 0,Y 352.757,Z 839.752,A -85,B 0,C 180,E1 16460.373,E2 16460.373} C_VEL
LIN {X 0,Y 352.82,Z 833.854,A -85,B 0,C 180,E1 16457.396,E2 16457.396} C_VEL
LIN {X 0,Y 353.289,Z 825.68,A -85,B 0,C 180,E1 16454.205,E2 16454.205} C_VEL
LIN {X 0,Y 354.283,Z 815.339,A -85,B 0,C 180,E1 16450.985,E2 16450.985} C_VEL
LIN {X 0,Y 355.795,Z 803.761,A -85,B 0,C 180,E1 16448.028,E2 16448.028} C_VEL
LIN {X 0,Y 357.865,Z 790.627,A -85,B 0,C 180,E1 16445.223,E2 16445.223} C_VEL
LIN {X 0,Y 360.427,Z 775.886,A -85,B 0,C 180,E1 16442.582,E2 16442.582} C_VEL
LIN {X 0,Y 363.45,Z 759.581,A -85,B 0,C 180,E1 16440.138,E2 16440.138} C_VEL
LIN {X 0,Y 366.634,Z 742.56,A -85,B 0,C 180,E1 16438.009,E2 16438.009} C_VEL
LIN {X 0,Y 369.877,Z 724.753,A -85,B 0,C 180,E1 16436.162,E2 16436.162} C_VEL
LIN {X 0,Y 373,Z 706.679,A -85,B 0,C 180,E1 16434.621,E2 16434.621} C_VEL
LIN {X 0,Y 376.096,Z 686.843,A -85,B 0,C 180,E1 16433.263,E2 16433.263} C_VEL
LIN {X 0,Y 378.966,Z 665.727,A -85,B 0,C 180,E1 16432.158,E2 16432.158} C_VEL
LIN {X 0,Y 381.256,Z 644.268,A -85,B 0,C 180,E1 16431.344,E2 16431.344} C_VEL
LIN {X 0,Y 382.618,Z 622.097,A -85,B 0,C 180,E1 16430.771,E2 16430.771} C_VEL
LIN {X 0,Y 390.111,Z 426.151,A -85,B 0,C 180,E1 16426.792,E2 16426.792} C_VEL
LIN {X 0,Y 386.551,Z 388.013,A -85,B 0,C 180,E1 16425.395,E2 16425.395} C_VEL
LIN {X 0,Y 381.69,Z 378.843,A -85,B 0,C 180,E1 16424.485,E2 16424.485} C_VEL
LIN {X 0,Y 375.097,Z 362.357,A -85,B 0,C 180,E1 16421.725,E2 16421.725} C_VEL
LIN {X 0,Y 367.882,Z 346.536,A -85,B 0,C 180,E1 16418.739,E2 16418.739} C_VEL
LIN {X 0,Y 362.108,Z 334.813,A -85,B 0,C 180,E1 16416.221,E2 16416.221} C_VEL
LIN {X 0,Y 358.372,Z 327.423,A -85,B 0,C 180,E1 16414.497,E2 16414.497} C_VEL
LIN {X 0,Y 355.641,Z 322.528,A -85,B 0,C 180,E1 16413.245,E2 16413.245} C_VEL
LIN {X 0,Y 353.897,Z 318.781,A -85,B 0,C 180,E1 16412.274,E2 16412.274} C_VEL
LIN {X 0,Y 353.829,Z 318.397,A -85,B 0,C 180,E1 16411.709,E2 16411.709} C_VEL
LIN {X 0,Y 353.827,Z 318.394,A -85,B 0,C 180,E1 16407.609,E2 16407.609} C_VEL
LIN {X 0,Y 353.824,Z 318.391,A -85,B 0,C 180,E1 16403.481,E2 16403.481} C_VEL
LIN {X 0,Y 353.819,Z 318.395,A -85,B 0,C 180,E1 16399.478,E2 16399.478} C_VEL
LIN {X 0,Y 353.817,Z 318.407,A -85,B 0,C 180,E1 16395.404,E2 16395.404} C_VEL
LIN {X 0,Y 353.816,Z 318.411,A -85,B 0,C 180,E1 16391.244,E2 16391.244} C_VEL
LIN {X 0,Y 353.812,Z 318.392,A -85,B 0,C 180,E1 16387.142,E2 16387.142} C_VEL
LIN {X 0,Y 353.807,Z 318.384,A -85,B 0,C 180,E1 16383.078,E2 16383.078} C_VEL
LIN {X 0,Y 353.807,Z 318.406,A -85,B 0,C 180,E1 16379.028,E2 16379.028} C_VEL
LIN {X 0,Y 353.816,Z 318.408,A -85,B 0,C 180,E1 16374.811,E2 16374.811} C_VEL
LIN {X 0,Y 353.818,Z 318.382,A -85,B 0,C 180,E1 16370.73,E2 16370.73} C_VEL
LIN {X 0,Y 353.83,Z 318.385,A -85,B 0,C 180,E1 16366.601,E2 16366.601} C_VEL
LIN {X 0,Y 353.845,Z 318.404,A -85,B 0,C 180,E1 16362.401,E2 16362.401} C_VEL
LIN {X 0,Y 353.855,Z 318.406,A -85,B 0,C 180,E1 16358.1,E2 16358.1} C_VEL
LIN {X 0,Y 353.841,Z 318.394,A -85,B 0,C 180,E1 16353.844,E2 16353.844} C_VEL
LIN {X 0,Y 353.843,Z 318.389,A -85,B 0,C 180,E1 16349.802,E2 16349.802} C_VEL
LIN {X 0,Y 353.847,Z 318.389,A -85,B 0,C 180,E1 16345.784,E2 16345.784} C_VEL
LIN {X 0,Y 353.854,Z 318.391,A -85,B 0,C 180,E1 16341.767,E2 16341.767} C_VEL
LIN {X 0,Y 353.858,Z 318.589,A -85,B 0,C 180,E1 16339.146,E2 16339.146} C_VEL
LIN {X 0,Y 355.214,Z 321.938,A -85,B 0,C 180,E1 16338.155,E2 16338.155} C_VEL
LIN {X 0,Y 356.194,Z 323.937,A -85,B 0,C 180,E1 16337.581,E2 16337.581} C_VEL
LIN {X 0,Y 359.806,Z 331.364,A -85,B 0,C 180,E1 16335.55,E2 16335.55} C_VEL
LIN {X 0,Y 365.113,Z 343.733,A -85,B 0,C 180,E1 16332.552,E2 16332.552} C_VEL
LIN {X 0,Y 367.193,Z 348.401,A -85,B 0,C 180,E1 16331.541,E2 16331.541} C_VEL
LIN {X 0,Y 379.033,Z 367.078,A -85,B 0,C 180,E1 16329.324,E2 16329.324} C_VEL
LIN {X 0,Y 389.575,Z 385.776,A -85,B 0,C 180,E1 16327.486,E2 16327.486} C_VEL
LIN {X 0,Y 384.372,Z 564.348,A -85,B 0,C 180,E1 16324.221,E2 16324.221} C_VEL
LIN {X 0,Y 383.473,Z 583.113,A -85,B 0,C 180,E1 16323.623,E2 16323.623} C_VEL
LIN {X 0,Y 382.001,Z 600.901,A -85,B 0,C 180,E1 16322.806,E2 16322.806} C_VEL
LIN {X 0,Y 380.036,Z 618.183,A -85,B 0,C 180,E1 16321.748,E2 16321.748} C_VEL
LIN {X 0,Y 377.634,Z 634.674,A -85,B 0,C 180,E1 16320.465,E2 16320.465} C_VEL
LIN {X 0,Y 374.767,Z 651.083,A -85,B 0,C 180,E1 16318.874,E2 16318.874} C_VEL
LIN {X 0,Y 371.677,Z 666.384,A -85,B 0,C 180,E1 16317.04,E2 16317.04} C_VEL
LIN {X 0,Y 368.609,Z 680.089,A -85,B 0,C 180,E1 16315.033,E2 16315.033} C_VEL
LIN {X 0,Y 365.431,Z 693.192,A -85,B 0,C 180,E1 16312.692,E2 16312.692} C_VEL
LIN {X 0,Y 362.5,Z 704.69,A -85,B 0,C 180,E1 16310.168,E2 16310.168} C_VEL
LIN {X 0,Y 359.935,Z 714.65,A -85,B 0,C 180,E1 16307.458,E2 16307.458} C_VEL
LIN {X 0,Y 357.763,Z 723.094,A -85,B 0,C 180,E1 16304.568,E2 16304.568} C_VEL
LIN {X 0,Y 356.161,Z 729.667,A -85,B 0,C 180,E1 16301.661,E2 16301.661} C_VEL
LIN {X 0,Y 355.001,Z 734.817,A -85,B 0,C 180,E1 16298.585,E2 16298.585} C_VEL
LIN {X 0,Y 354.248,Z 738.439,A -85,B 0,C 180,E1 16295.344,E2 16295.344} C_VEL
LIN {X 0,Y 353.897,Z 740.346,A -85,B 0,C 180,E1 16292.105,E2 16292.105} C_VEL
LIN {X 0,Y 353.848,Z 740.616,A -85,B 0,C 180,E1 16288.867,E2 16288.867} C_VEL
LIN {X 0,Y 353.866,Z 740.566,A -85,B 0,C 180,E1 16288.451,E2 16288.451} C_VEL
LIN {X 0,Y 352.976,Z 740.398,A -85,B 0,C 180,E1 16287.201,E2 16287.201} C_VEL
LIN {X 0,Y 348.515,Z 739.641,A -85,B 0,C 180,E1 16284.746,E2 16284.746} C_VEL
LIN {X 0,Y 346.754,Z 738.536,A -85,B 0,C 180,E1 16283.218,E2 16283.218} C_VEL
LIN {X 0,Y 346.714,Z 738.05,A -85,B 0,C 180,E1 16282.764,E2 16282.764} C_VEL
LIN {X 0,Y 347.737,Z 733.66,A -85,B 0,C 180,E1 16279.537,E2 16279.537} C_VEL
LIN {X 0,Y 349.321,Z 727.307,A -85,B 0,C 180,E1 16276.257,E2 16276.257} C_VEL
LIN {X 0,Y 351.36,Z 719.697,A -85,B 0,C 180,E1 16273.297,E2 16273.297} C_VEL
LIN {X 0,Y 353.982,Z 710.063,A -85,B 0,C 180,E1 16270.36,E2 16270.36} C_VEL
LIN {X 0,Y 356.844,Z 699.482,A -85,B 0,C 180,E1 16267.775,E2 16267.775} C_VEL
LIN {X 0,Y 359.992,Z 687.464,A -85,B 0,C 180,E1 16265.38,E2 16265.38} C_VEL
LIN {X 0,Y 363.293,Z 673.927,A -85,B 0,C 180,E1 16263.17,E2 16263.17} C_VEL
